// TwinCAT 3 PLC project TcoIo
// Title: TcoIo
// Company: Vortex.Library
// Author: Inxton
// ProjectVersion: 0.6.0.913
// ProgramVersion: 3.1.4023.0
// libraries:
//   Tc2_EtherCAT, * (Beckhoff Automation GmbH)
//   Tc2_Standard, * (Beckhoff Automation GmbH)
//   Tc2_System, * (Beckhoff Automation GmbH)
//   Tc3_Module, * (Beckhoff Automation GmbH)
//   TcoCore, 0.6.0.913 (Vortex.Library)
// project tree:
//   Diagnostics/EtherCAT/MasterDevice/Base/ EtcMasterBase_62654B43.TcDUT, SyncUnitsBase_AD6C35CE.TcDUT, SyncUnitTaskBase_FCD3CBF3.TcDUT, SyncUnitTasksBase_7C8711EB.TcDUT
//   Diagnostics/EtherCAT/MasterDevice/SyncUnit/ InfoData_8649EEEB.TcDUT, ITcoSyncUnit.TcIO, SyncUnitState.TcDUT, SyncUnitTask_AB2F5079.TcDUT, TcoSyncUnit.TcPOU
//   Diagnostics/EtherCAT/SlaveDevice/Base/ EtcSlaveBase_82538BE2.TcDUT, EtcSlaveBoxBase_77A0E4A7.TcDUT, EtcSlaveEndTerminalBase_866C7F0C.TcDUT, EtcSlaveTerminalBase_947E5A46.TcDUT
//   Diagnostics/EtherCAT/MasterDevice/ InfoData_84133AC9.TcDUT, Inputs_A65FACA4.TcDUT, Outputs_23C0ED1D.TcDUT, TcoEthercatDiagnosticsTask.TcPOU, TcoEthercatMasterDeviceState.TcDUT, ITcoEthercatMasterDevice.TcIO, TcoEthercatMasterDevice.TcPOU
//   Diagnostics/EtherCAT/MasterDevice/Messenger/ DiagnosticsMessenger.TcPOU, DiagnosticsMessengers.TcPOU
//   Diagnostics/EtherCAT/SlaveDevice/InfoData/ InfoData_23CBA837.TcDUT, InfoData_6F19DB2B.TcDUT
//   Diagnostics/EtherCAT/SlaveDevice/Inputs/ InputBase_8311D824.TcDUT
//   Diagnostics/EtherCAT/SlaveDevice/Outputs/ OutputBase_10CEE7DE.TcDUT
//   Diagnostics/EtherCAT/SlaveDevice/WcState/ WcState_0B2B16F9.TcDUT, WcState_9091E0EB.TcDUT
//   Diagnostics/EtherCAT/ TcoEthercat.TcGVL
//   Diagnostics/ProfinetComponent/ TcoPnIoComponent.TcPOU
//   EtherCAT/ eEcatState.TcDUT, eLinkState.TcDUT, ITcoEcatComponent.TcIO, TcoEcatSlaveState.TcPOU, TcoEcatComponent.TcPOU
//   / PlcTask.TcTTO
//   POUs/ MAIN.TcPOU
//   SpecialPlcTypes/ TcoAmsAddr.TcDUT, TcoAmsNetId.TcDUT
// real-time tasks:
//   TASK PlcTask: cycle T#10ms, priority 20, ADS port 350
//   TASK PlcTask1: cycle T#10ms, priority 21, ADS port 351
//   TASK PlcTask2: cycle T#10ms, priority 22, ADS port 352
// I/O:
//   DEVICE Device 1 (EtherCAT) (disabled), AmsNetId 172.20.10.104.2.1
//     Term 1 (EK1200) [EK1200-5000 EtherCAT Power supply (2A E-Bus)]
//       Term 2 (EL6002) [EL6002 Interface 2Ch. (RS232)]
//       Term 3 (EL1809) [EL1809 16Ch. Dig. Input 24V, 3ms]
//       Term 4 (EL2809) [EL2809 16Ch. Dig. Output 24V, 0.5A]
//       Term 5 (EL4004) [EL4004 4Ch. Ana. Output 0-10V, 12bit]
//       Term 6 (EL2809) [EL2809 16Ch. Dig. Output 24V, 0.5A]
//       Term 7 (EL6001) [EL6001 Interface (RS232)]
//       Term 8 (EL9011) [EL9011 End Terminal]
//   DEVICE Device 4 (EtherCAT) (disabled), AmsNetId 172.20.10.104.5.1
//     Term 9 (EK1100) [EK1100 EtherCAT Coupler (2A E-Bus)]
//       Term 10 (EK1122) [EK1122 2 port EtherCAT junction]
//         Term 11 (EK1100) [EK1100 EtherCAT Coupler (2A E-Bus)]
//           Term 12 (EL3174-0002) [EL3174-0002 4Ch. Ana. Input +/-10V, +/-20mA 16 Bit, Isolated Channels]
//           Term 13 (EL6001) [EL6001 Interface (RS232)]
//           Term 14 (EL3011) [EL3011 4Ch. Ana. Input 0-20mA DIFF]
//           Term 15 (EL2008) [EL2008 8Ch. Dig. Output 24V, 0.5A]
//           Term 16 (EL2008) [EL2008 8Ch. Dig. Output 24V, 0.5A]
//           Term 17 (EK1110) [EK1110 EtherCAT extension]
//         Term 18 (EK1100) [EK1100 EtherCAT Coupler (2A E-Bus)]
//           Term 19 (EL1809) [EL1809 16Ch. Dig. Input 24V, 3ms]
//           Term 20 (EL2809) [EL2809 16Ch. Dig. Output 24V, 0.5A]
//           Term 21 (EL1809) [EL1809 16Ch. Dig. Input 24V, 3ms]
//           Term 22 (EL3011) [EL3011 4Ch. Ana. Input 0-20mA DIFF]
//           Term 18 (EL9011) [EL9011 End Terminal]
//       Term 23 (EL3403) [EL3403 3Ch. Power Measuring]
//       Term 24 (EL6001) [EL6001 Interface (RS232)]
//       Term 25 (EL3024) [EL3024 4Ch. Ana. Input 4-20mA DIFF]
//       Term 19 (EL9011) [EL9011 End Terminal]
// variable links:
//   TcoIoTests/TcoIoTests Instance <-> Device 1 (EtherCAT)
//     PlcTask Inputs/GVL_iXlinker.Device_1_EtherCAT.InfoData.AmsNetId <-> InfoData/AmsNetId
//     PlcTask Inputs/GVL_iXlinker.Device_1_EtherCAT.InfoData.CfgSlaveCount <-> InfoData/CfgSlaveCount
//     PlcTask Inputs/GVL_iXlinker.Device_1_EtherCAT.InfoData.ChangeCount <-> InfoData/ChangeCount
//     PlcTask Inputs/GVL_iXlinker.Device_1_EtherCAT.InfoData.DevId <-> InfoData/DevId
//     PlcTask Inputs/GVL_iXlinker.Device_1_EtherCAT.Inputs.DevState <-> Inputs/DevState
//     PlcTask Inputs/GVL_iXlinker.Device_1_EtherCAT.Inputs.Frm0InputToggle <-> Inputs/Frm0InputToggle
//     PlcTask Inputs/GVL_iXlinker.Device_1_EtherCAT.Inputs.Frm0State <-> Inputs/Frm0State
//     PlcTask Inputs/GVL_iXlinker.Device_1_EtherCAT.Inputs.Frm0WcState <-> Inputs/Frm0WcState
//     PlcTask Inputs/GVL_iXlinker.Device_1_EtherCAT.Inputs.SlaveCount <-> Inputs/SlaveCount
//     PlcTask Inputs/GVL_iXlinker.Device_1_EtherCAT.SyncUnits._default.PlcTask1.InfoData.ObjectId <-> SyncUnits/<default>/PlcTask1/InfoData/ObjectId
//     PlcTask Inputs/GVL_iXlinker.Device_1_EtherCAT.SyncUnits._default.PlcTask1.InfoData.SlaveCount <-> SyncUnits/<default>/PlcTask1/InfoData/SlaveCount
//     PlcTask Inputs/GVL_iXlinker.Device_1_EtherCAT.SyncUnits._default.PlcTask1.InfoData.State <-> SyncUnits/<default>/PlcTask1/InfoData/State
//     PlcTask Inputs/GVL_iXlinker.Device_1_EtherCAT.SyncUnits._default.PlcTask1.WcState.WcState <-> SyncUnits/<default>/PlcTask1/WcState/WcState
//     PlcTask Outputs/GVL_iXlinker.Device_1_EtherCAT.Outputs.DevCtrl <-> Outputs/DevCtrl
//     PlcTask Outputs/GVL_iXlinker.Device_1_EtherCAT.Outputs.Frm0Ctrl <-> Outputs/Frm0Ctrl
//     PlcTask Outputs/GVL_iXlinker.Device_1_EtherCAT.Outputs.Frm0WcCtrl <-> Outputs/Frm0WcCtrl
//   TcoIoTests/TcoIoTests Instance <-> Device 1 (EtherCAT)/Term 1 (EK1200)/Term 2 (EL6002)
//     PlcTask Inputs/GVL_iXlinker.Device_1_EtherCAT.Term_1_EK1200.Term_2_EL6002.COM_TxPDO_Map_Inputs_Channel_1.Data_In[0] <-> COM TxPDO-Map Inputs Channel 1/Data In 0
//     PlcTask Inputs/GVL_iXlinker.Device_1_EtherCAT.Term_1_EK1200.Term_2_EL6002.COM_TxPDO_Map_Inputs_Channel_1.Data_In[10] <-> COM TxPDO-Map Inputs Channel 1/Data In 10
//     PlcTask Inputs/GVL_iXlinker.Device_1_EtherCAT.Term_1_EK1200.Term_2_EL6002.COM_TxPDO_Map_Inputs_Channel_1.Data_In[11] <-> COM TxPDO-Map Inputs Channel 1/Data In 11
//     PlcTask Inputs/GVL_iXlinker.Device_1_EtherCAT.Term_1_EK1200.Term_2_EL6002.COM_TxPDO_Map_Inputs_Channel_1.Data_In[12] <-> COM TxPDO-Map Inputs Channel 1/Data In 12
//     PlcTask Inputs/GVL_iXlinker.Device_1_EtherCAT.Term_1_EK1200.Term_2_EL6002.COM_TxPDO_Map_Inputs_Channel_1.Data_In[13] <-> COM TxPDO-Map Inputs Channel 1/Data In 13
//     PlcTask Inputs/GVL_iXlinker.Device_1_EtherCAT.Term_1_EK1200.Term_2_EL6002.COM_TxPDO_Map_Inputs_Channel_1.Data_In[14] <-> COM TxPDO-Map Inputs Channel 1/Data In 14
//     PlcTask Inputs/GVL_iXlinker.Device_1_EtherCAT.Term_1_EK1200.Term_2_EL6002.COM_TxPDO_Map_Inputs_Channel_1.Data_In[15] <-> COM TxPDO-Map Inputs Channel 1/Data In 15
//     PlcTask Inputs/GVL_iXlinker.Device_1_EtherCAT.Term_1_EK1200.Term_2_EL6002.COM_TxPDO_Map_Inputs_Channel_1.Data_In[16] <-> COM TxPDO-Map Inputs Channel 1/Data In 16
//     PlcTask Inputs/GVL_iXlinker.Device_1_EtherCAT.Term_1_EK1200.Term_2_EL6002.COM_TxPDO_Map_Inputs_Channel_1.Data_In[17] <-> COM TxPDO-Map Inputs Channel 1/Data In 17
//     PlcTask Inputs/GVL_iXlinker.Device_1_EtherCAT.Term_1_EK1200.Term_2_EL6002.COM_TxPDO_Map_Inputs_Channel_1.Data_In[18] <-> COM TxPDO-Map Inputs Channel 1/Data In 18
//     PlcTask Inputs/GVL_iXlinker.Device_1_EtherCAT.Term_1_EK1200.Term_2_EL6002.COM_TxPDO_Map_Inputs_Channel_1.Data_In[19] <-> COM TxPDO-Map Inputs Channel 1/Data In 19
//     PlcTask Inputs/GVL_iXlinker.Device_1_EtherCAT.Term_1_EK1200.Term_2_EL6002.COM_TxPDO_Map_Inputs_Channel_1.Data_In[1] <-> COM TxPDO-Map Inputs Channel 1/Data In 1
//     PlcTask Inputs/GVL_iXlinker.Device_1_EtherCAT.Term_1_EK1200.Term_2_EL6002.COM_TxPDO_Map_Inputs_Channel_1.Data_In[20] <-> COM TxPDO-Map Inputs Channel 1/Data In 20
//     PlcTask Inputs/GVL_iXlinker.Device_1_EtherCAT.Term_1_EK1200.Term_2_EL6002.COM_TxPDO_Map_Inputs_Channel_1.Data_In[21] <-> COM TxPDO-Map Inputs Channel 1/Data In 21
//     PlcTask Inputs/GVL_iXlinker.Device_1_EtherCAT.Term_1_EK1200.Term_2_EL6002.COM_TxPDO_Map_Inputs_Channel_1.Data_In[2] <-> COM TxPDO-Map Inputs Channel 1/Data In 2
//     PlcTask Inputs/GVL_iXlinker.Device_1_EtherCAT.Term_1_EK1200.Term_2_EL6002.COM_TxPDO_Map_Inputs_Channel_1.Data_In[3] <-> COM TxPDO-Map Inputs Channel 1/Data In 3
//     PlcTask Inputs/GVL_iXlinker.Device_1_EtherCAT.Term_1_EK1200.Term_2_EL6002.COM_TxPDO_Map_Inputs_Channel_1.Data_In[4] <-> COM TxPDO-Map Inputs Channel 1/Data In 4
//     PlcTask Inputs/GVL_iXlinker.Device_1_EtherCAT.Term_1_EK1200.Term_2_EL6002.COM_TxPDO_Map_Inputs_Channel_1.Data_In[5] <-> COM TxPDO-Map Inputs Channel 1/Data In 5
//     PlcTask Inputs/GVL_iXlinker.Device_1_EtherCAT.Term_1_EK1200.Term_2_EL6002.COM_TxPDO_Map_Inputs_Channel_1.Data_In[6] <-> COM TxPDO-Map Inputs Channel 1/Data In 6
//     PlcTask Inputs/GVL_iXlinker.Device_1_EtherCAT.Term_1_EK1200.Term_2_EL6002.COM_TxPDO_Map_Inputs_Channel_1.Data_In[7] <-> COM TxPDO-Map Inputs Channel 1/Data In 7
//     PlcTask Inputs/GVL_iXlinker.Device_1_EtherCAT.Term_1_EK1200.Term_2_EL6002.COM_TxPDO_Map_Inputs_Channel_1.Data_In[8] <-> COM TxPDO-Map Inputs Channel 1/Data In 8
//     PlcTask Inputs/GVL_iXlinker.Device_1_EtherCAT.Term_1_EK1200.Term_2_EL6002.COM_TxPDO_Map_Inputs_Channel_1.Data_In[9] <-> COM TxPDO-Map Inputs Channel 1/Data In 9
//     PlcTask Inputs/GVL_iXlinker.Device_1_EtherCAT.Term_1_EK1200.Term_2_EL6002.COM_TxPDO_Map_Inputs_Channel_2.Data_In[0] <-> COM TxPDO-Map Inputs Channel 2/Data In 0
//     PlcTask Inputs/GVL_iXlinker.Device_1_EtherCAT.Term_1_EK1200.Term_2_EL6002.COM_TxPDO_Map_Inputs_Channel_2.Data_In[10] <-> COM TxPDO-Map Inputs Channel 2/Data In 10
//     PlcTask Inputs/GVL_iXlinker.Device_1_EtherCAT.Term_1_EK1200.Term_2_EL6002.COM_TxPDO_Map_Inputs_Channel_2.Data_In[11] <-> COM TxPDO-Map Inputs Channel 2/Data In 11
//     PlcTask Inputs/GVL_iXlinker.Device_1_EtherCAT.Term_1_EK1200.Term_2_EL6002.COM_TxPDO_Map_Inputs_Channel_2.Data_In[12] <-> COM TxPDO-Map Inputs Channel 2/Data In 12
//     PlcTask Inputs/GVL_iXlinker.Device_1_EtherCAT.Term_1_EK1200.Term_2_EL6002.COM_TxPDO_Map_Inputs_Channel_2.Data_In[13] <-> COM TxPDO-Map Inputs Channel 2/Data In 13
//     PlcTask Inputs/GVL_iXlinker.Device_1_EtherCAT.Term_1_EK1200.Term_2_EL6002.COM_TxPDO_Map_Inputs_Channel_2.Data_In[14] <-> COM TxPDO-Map Inputs Channel 2/Data In 14
//     PlcTask Inputs/GVL_iXlinker.Device_1_EtherCAT.Term_1_EK1200.Term_2_EL6002.COM_TxPDO_Map_Inputs_Channel_2.Data_In[15] <-> COM TxPDO-Map Inputs Channel 2/Data In 15
//     PlcTask Inputs/GVL_iXlinker.Device_1_EtherCAT.Term_1_EK1200.Term_2_EL6002.COM_TxPDO_Map_Inputs_Channel_2.Data_In[16] <-> COM TxPDO-Map Inputs Channel 2/Data In 16
//     PlcTask Inputs/GVL_iXlinker.Device_1_EtherCAT.Term_1_EK1200.Term_2_EL6002.COM_TxPDO_Map_Inputs_Channel_2.Data_In[17] <-> COM TxPDO-Map Inputs Channel 2/Data In 17
//     PlcTask Inputs/GVL_iXlinker.Device_1_EtherCAT.Term_1_EK1200.Term_2_EL6002.COM_TxPDO_Map_Inputs_Channel_2.Data_In[18] <-> COM TxPDO-Map Inputs Channel 2/Data In 18
//     PlcTask Inputs/GVL_iXlinker.Device_1_EtherCAT.Term_1_EK1200.Term_2_EL6002.COM_TxPDO_Map_Inputs_Channel_2.Data_In[19] <-> COM TxPDO-Map Inputs Channel 2/Data In 19
//     PlcTask Inputs/GVL_iXlinker.Device_1_EtherCAT.Term_1_EK1200.Term_2_EL6002.COM_TxPDO_Map_Inputs_Channel_2.Data_In[1] <-> COM TxPDO-Map Inputs Channel 2/Data In 1
//     PlcTask Inputs/GVL_iXlinker.Device_1_EtherCAT.Term_1_EK1200.Term_2_EL6002.COM_TxPDO_Map_Inputs_Channel_2.Data_In[20] <-> COM TxPDO-Map Inputs Channel 2/Data In 20
//     PlcTask Inputs/GVL_iXlinker.Device_1_EtherCAT.Term_1_EK1200.Term_2_EL6002.COM_TxPDO_Map_Inputs_Channel_2.Data_In[21] <-> COM TxPDO-Map Inputs Channel 2/Data In 21
//     PlcTask Inputs/GVL_iXlinker.Device_1_EtherCAT.Term_1_EK1200.Term_2_EL6002.COM_TxPDO_Map_Inputs_Channel_2.Data_In[2] <-> COM TxPDO-Map Inputs Channel 2/Data In 2
//     PlcTask Inputs/GVL_iXlinker.Device_1_EtherCAT.Term_1_EK1200.Term_2_EL6002.COM_TxPDO_Map_Inputs_Channel_2.Data_In[3] <-> COM TxPDO-Map Inputs Channel 2/Data In 3
//     PlcTask Inputs/GVL_iXlinker.Device_1_EtherCAT.Term_1_EK1200.Term_2_EL6002.COM_TxPDO_Map_Inputs_Channel_2.Data_In[4] <-> COM TxPDO-Map Inputs Channel 2/Data In 4
//     PlcTask Inputs/GVL_iXlinker.Device_1_EtherCAT.Term_1_EK1200.Term_2_EL6002.COM_TxPDO_Map_Inputs_Channel_2.Data_In[5] <-> COM TxPDO-Map Inputs Channel 2/Data In 5
//     PlcTask Inputs/GVL_iXlinker.Device_1_EtherCAT.Term_1_EK1200.Term_2_EL6002.COM_TxPDO_Map_Inputs_Channel_2.Data_In[6] <-> COM TxPDO-Map Inputs Channel 2/Data In 6
//     PlcTask Inputs/GVL_iXlinker.Device_1_EtherCAT.Term_1_EK1200.Term_2_EL6002.COM_TxPDO_Map_Inputs_Channel_2.Data_In[7] <-> COM TxPDO-Map Inputs Channel 2/Data In 7
//     PlcTask Inputs/GVL_iXlinker.Device_1_EtherCAT.Term_1_EK1200.Term_2_EL6002.COM_TxPDO_Map_Inputs_Channel_2.Data_In[8] <-> COM TxPDO-Map Inputs Channel 2/Data In 8
//     PlcTask Inputs/GVL_iXlinker.Device_1_EtherCAT.Term_1_EK1200.Term_2_EL6002.COM_TxPDO_Map_Inputs_Channel_2.Data_In[9] <-> COM TxPDO-Map Inputs Channel 2/Data In 9
//     PlcTask Inputs/GVL_iXlinker.Device_1_EtherCAT.Term_1_EK1200.Term_2_EL6002.COM_TxPDO_Map_Inputs_Channel_1.Status/Buffer_full <-> COM TxPDO-Map Inputs Channel 1/Status/Buffer full
//     PlcTask Inputs/GVL_iXlinker.Device_1_EtherCAT.Term_1_EK1200.Term_2_EL6002.COM_TxPDO_Map_Inputs_Channel_2.Status/Buffer_full <-> COM TxPDO-Map Inputs Channel 2/Status/Buffer full
//     PlcTask Inputs/GVL_iXlinker.Device_1_EtherCAT.Term_1_EK1200.Term_2_EL6002.COM_TxPDO_Map_Inputs_Channel_1.Status/Framing_error <-> COM TxPDO-Map Inputs Channel 1/Status/Framing error
//     PlcTask Inputs/GVL_iXlinker.Device_1_EtherCAT.Term_1_EK1200.Term_2_EL6002.COM_TxPDO_Map_Inputs_Channel_2.Status/Framing_error <-> COM TxPDO-Map Inputs Channel 2/Status/Framing error
//     PlcTask Inputs/GVL_iXlinker.Device_1_EtherCAT.Term_1_EK1200.Term_2_EL6002.COM_TxPDO_Map_Inputs_Channel_1.Status/Init_accepted <-> COM TxPDO-Map Inputs Channel 1/Status/Init accepted
//     PlcTask Inputs/GVL_iXlinker.Device_1_EtherCAT.Term_1_EK1200.Term_2_EL6002.COM_TxPDO_Map_Inputs_Channel_2.Status/Init_accepted <-> COM TxPDO-Map Inputs Channel 2/Status/Init accepted
//     PlcTask Inputs/GVL_iXlinker.Device_1_EtherCAT.Term_1_EK1200.Term_2_EL6002.COM_TxPDO_Map_Inputs_Channel_1.Status/Input_length <-> COM TxPDO-Map Inputs Channel 1/Status/Input length
//     PlcTask Inputs/GVL_iXlinker.Device_1_EtherCAT.Term_1_EK1200.Term_2_EL6002.COM_TxPDO_Map_Inputs_Channel_2.Status/Input_length <-> COM TxPDO-Map Inputs Channel 2/Status/Input length
//     PlcTask Inputs/GVL_iXlinker.Device_1_EtherCAT.Term_1_EK1200.Term_2_EL6002.COM_TxPDO_Map_Inputs_Channel_1.Status/Overrun_error <-> COM TxPDO-Map Inputs Channel 1/Status/Overrun error
//     PlcTask Inputs/GVL_iXlinker.Device_1_EtherCAT.Term_1_EK1200.Term_2_EL6002.COM_TxPDO_Map_Inputs_Channel_2.Status/Overrun_error <-> COM TxPDO-Map Inputs Channel 2/Status/Overrun error
//     PlcTask Inputs/GVL_iXlinker.Device_1_EtherCAT.Term_1_EK1200.Term_2_EL6002.COM_TxPDO_Map_Inputs_Channel_1.Status/Parity_error <-> COM TxPDO-Map Inputs Channel 1/Status/Parity error
//     PlcTask Inputs/GVL_iXlinker.Device_1_EtherCAT.Term_1_EK1200.Term_2_EL6002.COM_TxPDO_Map_Inputs_Channel_2.Status/Parity_error <-> COM TxPDO-Map Inputs Channel 2/Status/Parity error
//     PlcTask Inputs/GVL_iXlinker.Device_1_EtherCAT.Term_1_EK1200.Term_2_EL6002.COM_TxPDO_Map_Inputs_Channel_1.Status/Receive_request <-> COM TxPDO-Map Inputs Channel 1/Status/Receive request
//     PlcTask Inputs/GVL_iXlinker.Device_1_EtherCAT.Term_1_EK1200.Term_2_EL6002.COM_TxPDO_Map_Inputs_Channel_2.Status/Receive_request <-> COM TxPDO-Map Inputs Channel 2/Status/Receive request
//     PlcTask Inputs/GVL_iXlinker.Device_1_EtherCAT.Term_1_EK1200.Term_2_EL6002.COM_TxPDO_Map_Inputs_Channel_1.Status/Transmit_accepted <-> COM TxPDO-Map Inputs Channel 1/Status/Transmit accepted
//     PlcTask Inputs/GVL_iXlinker.Device_1_EtherCAT.Term_1_EK1200.Term_2_EL6002.COM_TxPDO_Map_Inputs_Channel_2.Status/Transmit_accepted <-> COM TxPDO-Map Inputs Channel 2/Status/Transmit accepted
//     PlcTask Inputs/GVL_iXlinker.Device_1_EtherCAT.Term_1_EK1200.Term_2_EL6002.InfoData.AdsAddr <-> InfoData/AdsAddr
//     PlcTask Inputs/GVL_iXlinker.Device_1_EtherCAT.Term_1_EK1200.Term_2_EL6002.InfoData.State <-> InfoData/State
//     PlcTask Inputs/GVL_iXlinker.Device_1_EtherCAT.Term_1_EK1200.Term_2_EL6002.WcState.InputToggle <-> WcState/InputToggle
//     PlcTask Inputs/GVL_iXlinker.Device_1_EtherCAT.Term_1_EK1200.Term_2_EL6002.WcState.WcState <-> WcState/WcState
//     PlcTask Outputs/GVL_iXlinker.Device_1_EtherCAT.Term_1_EK1200.Term_2_EL6002.COM_RxPDO_Map_Outputs_Channel_1.Ctrl/Init_request <-> COM RxPDO-Map Outputs Channel 1/Ctrl/Init request
//     PlcTask Outputs/GVL_iXlinker.Device_1_EtherCAT.Term_1_EK1200.Term_2_EL6002.COM_RxPDO_Map_Outputs_Channel_2.Ctrl/Init_request <-> COM RxPDO-Map Outputs Channel 2/Ctrl/Init request
//     PlcTask Outputs/GVL_iXlinker.Device_1_EtherCAT.Term_1_EK1200.Term_2_EL6002.COM_RxPDO_Map_Outputs_Channel_1.Ctrl/Output_length <-> COM RxPDO-Map Outputs Channel 1/Ctrl/Output length
//     PlcTask Outputs/GVL_iXlinker.Device_1_EtherCAT.Term_1_EK1200.Term_2_EL6002.COM_RxPDO_Map_Outputs_Channel_2.Ctrl/Output_length <-> COM RxPDO-Map Outputs Channel 2/Ctrl/Output length
//     PlcTask Outputs/GVL_iXlinker.Device_1_EtherCAT.Term_1_EK1200.Term_2_EL6002.COM_RxPDO_Map_Outputs_Channel_1.Ctrl/Receive_accepted <-> COM RxPDO-Map Outputs Channel 1/Ctrl/Receive accepted
//     PlcTask Outputs/GVL_iXlinker.Device_1_EtherCAT.Term_1_EK1200.Term_2_EL6002.COM_RxPDO_Map_Outputs_Channel_2.Ctrl/Receive_accepted <-> COM RxPDO-Map Outputs Channel 2/Ctrl/Receive accepted
//     PlcTask Outputs/GVL_iXlinker.Device_1_EtherCAT.Term_1_EK1200.Term_2_EL6002.COM_RxPDO_Map_Outputs_Channel_1.Ctrl/Send_continuous <-> COM RxPDO-Map Outputs Channel 1/Ctrl/Send continuous
//     PlcTask Outputs/GVL_iXlinker.Device_1_EtherCAT.Term_1_EK1200.Term_2_EL6002.COM_RxPDO_Map_Outputs_Channel_2.Ctrl/Send_continuous <-> COM RxPDO-Map Outputs Channel 2/Ctrl/Send continuous
//     PlcTask Outputs/GVL_iXlinker.Device_1_EtherCAT.Term_1_EK1200.Term_2_EL6002.COM_RxPDO_Map_Outputs_Channel_1.Ctrl/Transmit_request <-> COM RxPDO-Map Outputs Channel 1/Ctrl/Transmit request
//     PlcTask Outputs/GVL_iXlinker.Device_1_EtherCAT.Term_1_EK1200.Term_2_EL6002.COM_RxPDO_Map_Outputs_Channel_2.Ctrl/Transmit_request <-> COM RxPDO-Map Outputs Channel 2/Ctrl/Transmit request
//     PlcTask Outputs/GVL_iXlinker.Device_1_EtherCAT.Term_1_EK1200.Term_2_EL6002.COM_RxPDO_Map_Outputs_Channel_1.Data_Out[0] <-> COM RxPDO-Map Outputs Channel 1/Data Out 0
//     PlcTask Outputs/GVL_iXlinker.Device_1_EtherCAT.Term_1_EK1200.Term_2_EL6002.COM_RxPDO_Map_Outputs_Channel_1.Data_Out[10] <-> COM RxPDO-Map Outputs Channel 1/Data Out 10
//     PlcTask Outputs/GVL_iXlinker.Device_1_EtherCAT.Term_1_EK1200.Term_2_EL6002.COM_RxPDO_Map_Outputs_Channel_1.Data_Out[11] <-> COM RxPDO-Map Outputs Channel 1/Data Out 11
//     PlcTask Outputs/GVL_iXlinker.Device_1_EtherCAT.Term_1_EK1200.Term_2_EL6002.COM_RxPDO_Map_Outputs_Channel_1.Data_Out[12] <-> COM RxPDO-Map Outputs Channel 1/Data Out 12
//     PlcTask Outputs/GVL_iXlinker.Device_1_EtherCAT.Term_1_EK1200.Term_2_EL6002.COM_RxPDO_Map_Outputs_Channel_1.Data_Out[13] <-> COM RxPDO-Map Outputs Channel 1/Data Out 13
//     PlcTask Outputs/GVL_iXlinker.Device_1_EtherCAT.Term_1_EK1200.Term_2_EL6002.COM_RxPDO_Map_Outputs_Channel_1.Data_Out[14] <-> COM RxPDO-Map Outputs Channel 1/Data Out 14
//     PlcTask Outputs/GVL_iXlinker.Device_1_EtherCAT.Term_1_EK1200.Term_2_EL6002.COM_RxPDO_Map_Outputs_Channel_1.Data_Out[15] <-> COM RxPDO-Map Outputs Channel 1/Data Out 15
//     PlcTask Outputs/GVL_iXlinker.Device_1_EtherCAT.Term_1_EK1200.Term_2_EL6002.COM_RxPDO_Map_Outputs_Channel_1.Data_Out[16] <-> COM RxPDO-Map Outputs Channel 1/Data Out 16
//     PlcTask Outputs/GVL_iXlinker.Device_1_EtherCAT.Term_1_EK1200.Term_2_EL6002.COM_RxPDO_Map_Outputs_Channel_1.Data_Out[17] <-> COM RxPDO-Map Outputs Channel 1/Data Out 17
//     PlcTask Outputs/GVL_iXlinker.Device_1_EtherCAT.Term_1_EK1200.Term_2_EL6002.COM_RxPDO_Map_Outputs_Channel_1.Data_Out[18] <-> COM RxPDO-Map Outputs Channel 1/Data Out 18
//     PlcTask Outputs/GVL_iXlinker.Device_1_EtherCAT.Term_1_EK1200.Term_2_EL6002.COM_RxPDO_Map_Outputs_Channel_1.Data_Out[19] <-> COM RxPDO-Map Outputs Channel 1/Data Out 19
//     PlcTask Outputs/GVL_iXlinker.Device_1_EtherCAT.Term_1_EK1200.Term_2_EL6002.COM_RxPDO_Map_Outputs_Channel_1.Data_Out[1] <-> COM RxPDO-Map Outputs Channel 1/Data Out 1
//     PlcTask Outputs/GVL_iXlinker.Device_1_EtherCAT.Term_1_EK1200.Term_2_EL6002.COM_RxPDO_Map_Outputs_Channel_1.Data_Out[20] <-> COM RxPDO-Map Outputs Channel 1/Data Out 20
//     PlcTask Outputs/GVL_iXlinker.Device_1_EtherCAT.Term_1_EK1200.Term_2_EL6002.COM_RxPDO_Map_Outputs_Channel_1.Data_Out[21] <-> COM RxPDO-Map Outputs Channel 1/Data Out 21
//     PlcTask Outputs/GVL_iXlinker.Device_1_EtherCAT.Term_1_EK1200.Term_2_EL6002.COM_RxPDO_Map_Outputs_Channel_1.Data_Out[2] <-> COM RxPDO-Map Outputs Channel 1/Data Out 2
//     PlcTask Outputs/GVL_iXlinker.Device_1_EtherCAT.Term_1_EK1200.Term_2_EL6002.COM_RxPDO_Map_Outputs_Channel_1.Data_Out[3] <-> COM RxPDO-Map Outputs Channel 1/Data Out 3
//     PlcTask Outputs/GVL_iXlinker.Device_1_EtherCAT.Term_1_EK1200.Term_2_EL6002.COM_RxPDO_Map_Outputs_Channel_1.Data_Out[4] <-> COM RxPDO-Map Outputs Channel 1/Data Out 4
//     PlcTask Outputs/GVL_iXlinker.Device_1_EtherCAT.Term_1_EK1200.Term_2_EL6002.COM_RxPDO_Map_Outputs_Channel_1.Data_Out[5] <-> COM RxPDO-Map Outputs Channel 1/Data Out 5
//     PlcTask Outputs/GVL_iXlinker.Device_1_EtherCAT.Term_1_EK1200.Term_2_EL6002.COM_RxPDO_Map_Outputs_Channel_1.Data_Out[6] <-> COM RxPDO-Map Outputs Channel 1/Data Out 6
//     PlcTask Outputs/GVL_iXlinker.Device_1_EtherCAT.Term_1_EK1200.Term_2_EL6002.COM_RxPDO_Map_Outputs_Channel_1.Data_Out[7] <-> COM RxPDO-Map Outputs Channel 1/Data Out 7
//     PlcTask Outputs/GVL_iXlinker.Device_1_EtherCAT.Term_1_EK1200.Term_2_EL6002.COM_RxPDO_Map_Outputs_Channel_1.Data_Out[8] <-> COM RxPDO-Map Outputs Channel 1/Data Out 8
//     PlcTask Outputs/GVL_iXlinker.Device_1_EtherCAT.Term_1_EK1200.Term_2_EL6002.COM_RxPDO_Map_Outputs_Channel_1.Data_Out[9] <-> COM RxPDO-Map Outputs Channel 1/Data Out 9
//     PlcTask Outputs/GVL_iXlinker.Device_1_EtherCAT.Term_1_EK1200.Term_2_EL6002.COM_RxPDO_Map_Outputs_Channel_2.Data_Out[0] <-> COM RxPDO-Map Outputs Channel 2/Data Out 0
//     PlcTask Outputs/GVL_iXlinker.Device_1_EtherCAT.Term_1_EK1200.Term_2_EL6002.COM_RxPDO_Map_Outputs_Channel_2.Data_Out[10] <-> COM RxPDO-Map Outputs Channel 2/Data Out 10
//     PlcTask Outputs/GVL_iXlinker.Device_1_EtherCAT.Term_1_EK1200.Term_2_EL6002.COM_RxPDO_Map_Outputs_Channel_2.Data_Out[11] <-> COM RxPDO-Map Outputs Channel 2/Data Out 11
//     PlcTask Outputs/GVL_iXlinker.Device_1_EtherCAT.Term_1_EK1200.Term_2_EL6002.COM_RxPDO_Map_Outputs_Channel_2.Data_Out[12] <-> COM RxPDO-Map Outputs Channel 2/Data Out 12
//     PlcTask Outputs/GVL_iXlinker.Device_1_EtherCAT.Term_1_EK1200.Term_2_EL6002.COM_RxPDO_Map_Outputs_Channel_2.Data_Out[13] <-> COM RxPDO-Map Outputs Channel 2/Data Out 13
//     PlcTask Outputs/GVL_iXlinker.Device_1_EtherCAT.Term_1_EK1200.Term_2_EL6002.COM_RxPDO_Map_Outputs_Channel_2.Data_Out[14] <-> COM RxPDO-Map Outputs Channel 2/Data Out 14
//     PlcTask Outputs/GVL_iXlinker.Device_1_EtherCAT.Term_1_EK1200.Term_2_EL6002.COM_RxPDO_Map_Outputs_Channel_2.Data_Out[15] <-> COM RxPDO-Map Outputs Channel 2/Data Out 15
//     PlcTask Outputs/GVL_iXlinker.Device_1_EtherCAT.Term_1_EK1200.Term_2_EL6002.COM_RxPDO_Map_Outputs_Channel_2.Data_Out[16] <-> COM RxPDO-Map Outputs Channel 2/Data Out 16
//     PlcTask Outputs/GVL_iXlinker.Device_1_EtherCAT.Term_1_EK1200.Term_2_EL6002.COM_RxPDO_Map_Outputs_Channel_2.Data_Out[17] <-> COM RxPDO-Map Outputs Channel 2/Data Out 17
//     PlcTask Outputs/GVL_iXlinker.Device_1_EtherCAT.Term_1_EK1200.Term_2_EL6002.COM_RxPDO_Map_Outputs_Channel_2.Data_Out[18] <-> COM RxPDO-Map Outputs Channel 2/Data Out 18
//     PlcTask Outputs/GVL_iXlinker.Device_1_EtherCAT.Term_1_EK1200.Term_2_EL6002.COM_RxPDO_Map_Outputs_Channel_2.Data_Out[19] <-> COM RxPDO-Map Outputs Channel 2/Data Out 19
//     PlcTask Outputs/GVL_iXlinker.Device_1_EtherCAT.Term_1_EK1200.Term_2_EL6002.COM_RxPDO_Map_Outputs_Channel_2.Data_Out[1] <-> COM RxPDO-Map Outputs Channel 2/Data Out 1
//     PlcTask Outputs/GVL_iXlinker.Device_1_EtherCAT.Term_1_EK1200.Term_2_EL6002.COM_RxPDO_Map_Outputs_Channel_2.Data_Out[20] <-> COM RxPDO-Map Outputs Channel 2/Data Out 20
//     PlcTask Outputs/GVL_iXlinker.Device_1_EtherCAT.Term_1_EK1200.Term_2_EL6002.COM_RxPDO_Map_Outputs_Channel_2.Data_Out[21] <-> COM RxPDO-Map Outputs Channel 2/Data Out 21
//     PlcTask Outputs/GVL_iXlinker.Device_1_EtherCAT.Term_1_EK1200.Term_2_EL6002.COM_RxPDO_Map_Outputs_Channel_2.Data_Out[2] <-> COM RxPDO-Map Outputs Channel 2/Data Out 2
//     PlcTask Outputs/GVL_iXlinker.Device_1_EtherCAT.Term_1_EK1200.Term_2_EL6002.COM_RxPDO_Map_Outputs_Channel_2.Data_Out[3] <-> COM RxPDO-Map Outputs Channel 2/Data Out 3
//     PlcTask Outputs/GVL_iXlinker.Device_1_EtherCAT.Term_1_EK1200.Term_2_EL6002.COM_RxPDO_Map_Outputs_Channel_2.Data_Out[4] <-> COM RxPDO-Map Outputs Channel 2/Data Out 4
//     PlcTask Outputs/GVL_iXlinker.Device_1_EtherCAT.Term_1_EK1200.Term_2_EL6002.COM_RxPDO_Map_Outputs_Channel_2.Data_Out[5] <-> COM RxPDO-Map Outputs Channel 2/Data Out 5
//     PlcTask Outputs/GVL_iXlinker.Device_1_EtherCAT.Term_1_EK1200.Term_2_EL6002.COM_RxPDO_Map_Outputs_Channel_2.Data_Out[6] <-> COM RxPDO-Map Outputs Channel 2/Data Out 6
//     PlcTask Outputs/GVL_iXlinker.Device_1_EtherCAT.Term_1_EK1200.Term_2_EL6002.COM_RxPDO_Map_Outputs_Channel_2.Data_Out[7] <-> COM RxPDO-Map Outputs Channel 2/Data Out 7
//     PlcTask Outputs/GVL_iXlinker.Device_1_EtherCAT.Term_1_EK1200.Term_2_EL6002.COM_RxPDO_Map_Outputs_Channel_2.Data_Out[8] <-> COM RxPDO-Map Outputs Channel 2/Data Out 8
//     PlcTask Outputs/GVL_iXlinker.Device_1_EtherCAT.Term_1_EK1200.Term_2_EL6002.COM_RxPDO_Map_Outputs_Channel_2.Data_Out[9] <-> COM RxPDO-Map Outputs Channel 2/Data Out 9
//   TcoIoTests/TcoIoTests Instance <-> Device 1 (EtherCAT)/Term 1 (EK1200)/Term 3 (EL1809)
//     PlcTask Inputs/GVL_iXlinker.Device_1_EtherCAT.Term_1_EK1200.Term_3_EL1809.Channel_{1..16}.Input <-> Channel {1..16}/Input  (16 links)
//     PlcTask Inputs/GVL_iXlinker.Device_1_EtherCAT.Term_1_EK1200.Term_3_EL1809.InfoData.State <-> InfoData/State
//     PlcTask Inputs/GVL_iXlinker.Device_1_EtherCAT.Term_1_EK1200.Term_3_EL1809.WcState.InputToggle <-> WcState/InputToggle
//     PlcTask Inputs/GVL_iXlinker.Device_1_EtherCAT.Term_1_EK1200.Term_3_EL1809.WcState.WcState <-> WcState/WcState
//   TcoIoTests/TcoIoTests Instance <-> Device 1 (EtherCAT)/Term 1 (EK1200)/Term 4 (EL2809)
//     PlcTask Inputs/GVL_iXlinker.Device_1_EtherCAT.Term_1_EK1200.Term_4_EL2809.InfoData.State <-> InfoData/State
//     PlcTask Inputs/GVL_iXlinker.Device_1_EtherCAT.Term_1_EK1200.Term_4_EL2809.WcState.WcState <-> WcState/WcState
//     PlcTask Outputs/GVL_iXlinker.Device_1_EtherCAT.Term_1_EK1200.Term_4_EL2809.Channel_{1..16}.Output <-> Channel {1..16}/Output  (16 links)
//   TcoIoTests/TcoIoTests Instance <-> Device 1 (EtherCAT)/Term 1 (EK1200)/Term 5 (EL4004)
//     PlcTask Inputs/GVL_iXlinker.Device_1_EtherCAT.Term_1_EK1200.Term_5_EL4004.InfoData.AdsAddr <-> InfoData/AdsAddr
//     PlcTask Inputs/GVL_iXlinker.Device_1_EtherCAT.Term_1_EK1200.Term_5_EL4004.InfoData.State <-> InfoData/State
//     PlcTask Inputs/GVL_iXlinker.Device_1_EtherCAT.Term_1_EK1200.Term_5_EL4004.WcState.WcState <-> WcState/WcState
//     PlcTask Outputs/GVL_iXlinker.Device_1_EtherCAT.Term_1_EK1200.Term_5_EL4004.AO_Outputs_Channel_{1..4}.Analog_output <-> AO Outputs Channel {1..4}/Analog output  (4 links)
//   TcoIoTests/TcoIoTests Instance <-> Device 1 (EtherCAT)/Term 1 (EK1200)/Term 6 (EL2809)
//     PlcTask Inputs/GVL_iXlinker.Device_1_EtherCAT.Term_1_EK1200.Term_6_EL2809.InfoData.State <-> InfoData/State
//     PlcTask Inputs/GVL_iXlinker.Device_1_EtherCAT.Term_1_EK1200.Term_6_EL2809.WcState.WcState <-> WcState/WcState
//     PlcTask Outputs/GVL_iXlinker.Device_1_EtherCAT.Term_1_EK1200.Term_6_EL2809.Channel_{1..16}.Output <-> Channel {1..16}/Output  (16 links)
//   TcoIoTests/TcoIoTests Instance <-> Device 1 (EtherCAT)/Term 1 (EK1200)/Term 7 (EL6001)
//     PlcTask Inputs/GVL_iXlinker.Device_1_EtherCAT.Term_1_EK1200.Term_7_EL6001.COM_Inputs.Data_In[{0..21}] <-> COM Inputs/Data In {0..21}  (22 links)
//     PlcTask Inputs/GVL_iXlinker.Device_1_EtherCAT.Term_1_EK1200.Term_7_EL6001.COM_Inputs.Status/Buffer_full <-> COM Inputs/Status/Buffer full
//     PlcTask Inputs/GVL_iXlinker.Device_1_EtherCAT.Term_1_EK1200.Term_7_EL6001.COM_Inputs.Status/Framing_error <-> COM Inputs/Status/Framing error
//     PlcTask Inputs/GVL_iXlinker.Device_1_EtherCAT.Term_1_EK1200.Term_7_EL6001.COM_Inputs.Status/Init_accepted <-> COM Inputs/Status/Init accepted
//     PlcTask Inputs/GVL_iXlinker.Device_1_EtherCAT.Term_1_EK1200.Term_7_EL6001.COM_Inputs.Status/Input_length <-> COM Inputs/Status/Input length
//     PlcTask Inputs/GVL_iXlinker.Device_1_EtherCAT.Term_1_EK1200.Term_7_EL6001.COM_Inputs.Status/Overrun_error <-> COM Inputs/Status/Overrun error
//     PlcTask Inputs/GVL_iXlinker.Device_1_EtherCAT.Term_1_EK1200.Term_7_EL6001.COM_Inputs.Status/Parity_error <-> COM Inputs/Status/Parity error
//     PlcTask Inputs/GVL_iXlinker.Device_1_EtherCAT.Term_1_EK1200.Term_7_EL6001.COM_Inputs.Status/Receive_request <-> COM Inputs/Status/Receive request
//     PlcTask Inputs/GVL_iXlinker.Device_1_EtherCAT.Term_1_EK1200.Term_7_EL6001.COM_Inputs.Status/Transmit_accepted <-> COM Inputs/Status/Transmit accepted
//     PlcTask Inputs/GVL_iXlinker.Device_1_EtherCAT.Term_1_EK1200.Term_7_EL6001.InfoData.AdsAddr <-> InfoData/AdsAddr
//     PlcTask Inputs/GVL_iXlinker.Device_1_EtherCAT.Term_1_EK1200.Term_7_EL6001.InfoData.State <-> InfoData/State
//     PlcTask Inputs/GVL_iXlinker.Device_1_EtherCAT.Term_1_EK1200.Term_7_EL6001.WcState.InputToggle <-> WcState/InputToggle
//     PlcTask Inputs/GVL_iXlinker.Device_1_EtherCAT.Term_1_EK1200.Term_7_EL6001.WcState.WcState <-> WcState/WcState
//     PlcTask Outputs/GVL_iXlinker.Device_1_EtherCAT.Term_1_EK1200.Term_7_EL6001.COM_Outputs.Ctrl/Init_request <-> COM Outputs/Ctrl/Init request
//     PlcTask Outputs/GVL_iXlinker.Device_1_EtherCAT.Term_1_EK1200.Term_7_EL6001.COM_Outputs.Ctrl/Output_length <-> COM Outputs/Ctrl/Output length
//     PlcTask Outputs/GVL_iXlinker.Device_1_EtherCAT.Term_1_EK1200.Term_7_EL6001.COM_Outputs.Ctrl/Receive_accepted <-> COM Outputs/Ctrl/Receive accepted
//     PlcTask Outputs/GVL_iXlinker.Device_1_EtherCAT.Term_1_EK1200.Term_7_EL6001.COM_Outputs.Ctrl/Send_continues <-> COM Outputs/Ctrl/Send continues
//     PlcTask Outputs/GVL_iXlinker.Device_1_EtherCAT.Term_1_EK1200.Term_7_EL6001.COM_Outputs.Ctrl/Transmit_request <-> COM Outputs/Ctrl/Transmit request
//     PlcTask Outputs/GVL_iXlinker.Device_1_EtherCAT.Term_1_EK1200.Term_7_EL6001.COM_Outputs.Data_Out[{0..21}] <-> COM Outputs/Data Out {0..21}  (22 links)
//   TcoIoTests/TcoIoTests Instance <-> Device 4 (EtherCAT)
//     PlcTask Inputs/GVL_iXlinker.Device_4_EtherCAT.InfoData.AmsNetId <-> InfoData/AmsNetId
//     PlcTask Inputs/GVL_iXlinker.Device_4_EtherCAT.InfoData.CfgSlaveCount <-> InfoData/CfgSlaveCount
//     PlcTask Inputs/GVL_iXlinker.Device_4_EtherCAT.InfoData.ChangeCount <-> InfoData/ChangeCount
//     PlcTask Inputs/GVL_iXlinker.Device_4_EtherCAT.InfoData.DevId <-> InfoData/DevId
//     PlcTask Inputs/GVL_iXlinker.Device_4_EtherCAT.Inputs.DevState <-> Inputs/DevState
//     PlcTask Inputs/GVL_iXlinker.Device_4_EtherCAT.Inputs.Frm0InputToggle <-> Inputs/Frm0InputToggle
//     PlcTask Inputs/GVL_iXlinker.Device_4_EtherCAT.Inputs.Frm0State <-> Inputs/Frm0State
//     PlcTask Inputs/GVL_iXlinker.Device_4_EtherCAT.Inputs.Frm0WcState <-> Inputs/Frm0WcState
//     PlcTask Inputs/GVL_iXlinker.Device_4_EtherCAT.Inputs.SlaveCount <-> Inputs/SlaveCount
//     PlcTask Outputs/GVL_iXlinker.Device_4_EtherCAT.Outputs.DevCtrl <-> Outputs/DevCtrl
//     PlcTask Outputs/GVL_iXlinker.Device_4_EtherCAT.Outputs.Frm0Ctrl <-> Outputs/Frm0Ctrl
//     PlcTask Outputs/GVL_iXlinker.Device_4_EtherCAT.Outputs.Frm0WcCtrl <-> Outputs/Frm0WcCtrl
//   TcoIoTests/TcoIoTests Instance <-> Device 4 (EtherCAT)/Term 9 (EK1100)
//     PlcTask Inputs/GVL_iXlinker.Device_4_EtherCAT.Term_9_EK1100.InfoData.State <-> InfoData/State

CONFIGURATION TcoIo
    RESOURCE PLC ON TwinCAT3
        TASK PlcTask(INTERVAL := T#15ms, PRIORITY := 12);
        PROGRAM MAIN WITH PlcTask : MAIN;
    END_RESOURCE
END_CONFIGURATION

// ---- Diagnostics/EtherCAT/MasterDevice/Base/EtcMasterBase_62654B43.TcDUT
TYPE EtcMasterBase_62654B43 :
STRUCT
END_STRUCT
END_TYPE

// ---- Diagnostics/EtherCAT/MasterDevice/Base/SyncUnitsBase_AD6C35CE.TcDUT
TYPE SyncUnitsBase_AD6C35CE :
STRUCT
END_STRUCT
END_TYPE

// ---- Diagnostics/EtherCAT/MasterDevice/Base/SyncUnitTaskBase_FCD3CBF3.TcDUT
TYPE SyncUnitTaskBase_FCD3CBF3 :
STRUCT
END_STRUCT
END_TYPE

// ---- Diagnostics/EtherCAT/MasterDevice/Base/SyncUnitTasksBase_7C8711EB.TcDUT
TYPE SyncUnitTasksBase_7C8711EB :
STRUCT
END_STRUCT
END_TYPE

// ---- Diagnostics/EtherCAT/MasterDevice/SyncUnit/InfoData_8649EEEB.TcDUT
{attribute 'GeneratedUsingTerminal: IODEVICETYPE_ETHERCATPROT'}
{attribute addProperty BoxType "IODEVICETYPE_ETHERCATPROT"}
{attribute addProperty Id "ObjectIdAT %I*DWORD4StateAT %I*UINT2SlaveCountAT %I*UINT2"}
{attribute addProperty CRC "2252992235"}
{attribute addProperty Size "8"}
TYPE InfoData_8649EEEB :
STRUCT
    {attribute addProperty Name "ObjectId"}
    ObjectId AT %I* : DWORD;
    {attribute addProperty Name "State"}
    State AT %I* : UINT;
    {attribute addProperty Name "SlaveCount"}
    SlaveCount AT %I* : UINT;
END_STRUCT
END_TYPE

// ---- Diagnostics/EtherCAT/MasterDevice/SyncUnit/SyncUnitState.TcDUT
TYPE SyncUnitState : 
STRUCT
    {attribute addProperty Name "At least one slave in 'INIT' state"}
    AtLeastOneSlaveInInitState : BOOL;
    {attribute addProperty Name "At least one slave in 'PREOP' state"}
    AtLeastOneSlaveInPreopState : BOOL;
    {attribute addProperty Name "At least one slave in 'BOOT' state"}
    AtLeastOneSlaveInBootState : BOOL;
    {attribute addProperty Name "At least one slave in 'SAFEOP' state"}
    AtLeastOneSlaveInSafeOpState : BOOL;
    {attribute addProperty Name "At least one slave in 'OP' state"}
    AtLeastOneSlaveInOpState : BOOL;
    {attribute addProperty Name "At least one slave signals error"}
    AtLeastOneSlaveSignalsError : BOOL;
    {attribute addProperty Name "Invalid vendorId, productCode... read"}
    InvalidVendoridOrProductcodeRead : BOOL;
    {attribute addProperty Name "Initialization error occurred"}
    InitializationErrorOccurred : BOOL;
    {attribute addProperty Name "At least one slave disabled"}
    AtLeastOneSlaveDisabled : BOOL;
    {attribute addProperty Name "At least one slave not present"}
    AtLeastOneSlaveNotPresent : BOOL;
    {attribute addProperty Name "At least one slave signals link error"}
    AtLeastOneSlaveSignalsLinkError : BOOL;
    {attribute addProperty Name "At least one slave signals missing link"}
    AtLeastOneSlaveSignalsMissingLink : BOOL;
    {attribute addProperty Name "At least one slave signals unexpected link"}
    AtLeastOneSlaveSignalsUnexpectedLink : BOOL;
END_STRUCT
END_TYPE

// ---- Diagnostics/EtherCAT/MasterDevice/SyncUnit/SyncUnitTask_AB2F5079.TcDUT
{attribute 'GeneratedUsingTerminal: IODEVICETYPE_ETHERCATPROT'}
{attribute addProperty BoxType "IODEVICETYPE_ETHERCATPROT"}
{attribute addProperty Id "WcStateAT %I*WcState_0B2B16F91InfoDataAT %I*InfoData_8649EEEB8"}
{attribute addProperty CRC "2872004729"}
{attribute addProperty Size "9"}
TYPE SyncUnitTask_AB2F5079 EXTENDS SyncUnitTaskBase_FCD3CBF3 :
STRUCT
    {attribute addProperty Name "WcState"}
    WcState : WcState_0B2B16F9;
    {attribute addProperty Name "InfoData"}
    InfoData : InfoData_8649EEEB;
END_STRUCT
END_TYPE

// ---- Diagnostics/EtherCAT/SlaveDevice/Base/EtcSlaveBase_82538BE2.TcDUT
TYPE EtcSlaveBase_82538BE2 :
STRUCT
END_STRUCT
END_TYPE

// ---- Diagnostics/EtherCAT/SlaveDevice/Base/EtcSlaveBoxBase_77A0E4A7.TcDUT
{attribute clr[Container(Layout.Stack)]}
{attribute clr[Group(Layout.GroupBox)]}
{attribute addProperty PreviousPort "Unknown"}
{attribute addProperty SyncUnit "Unknown"}
TYPE EtcSlaveBoxBase_77A0E4A7 EXTENDS EtcSlaveBase_82538BE2 :
STRUCT
END_STRUCT
END_TYPE

// ---- Diagnostics/EtherCAT/SlaveDevice/Base/EtcSlaveEndTerminalBase_866C7F0C.TcDUT
{attribute clr[Container(Layout.Stack)]}
{attribute clr[Group(Layout.GroupBox)]}
{attribute addProperty PreviousPort "Unknown"}
{attribute addProperty SyncUnit "Unknown"}
TYPE EtcSlaveEndTerminalBase_866C7F0C EXTENDS EtcSlaveBase_82538BE2 :
STRUCT
END_STRUCT
END_TYPE

// ---- Diagnostics/EtherCAT/SlaveDevice/Base/EtcSlaveTerminalBase_947E5A46.TcDUT
{attribute clr[Container(Layout.Stack)]}
{attribute clr[Group(Layout.GroupBox)]}
{attribute addProperty PreviousPort "Unknown"}
{attribute addProperty SyncUnit "Unknown"}
TYPE EtcSlaveTerminalBase_947E5A46 EXTENDS EtcSlaveBase_82538BE2 :
STRUCT
END_STRUCT
END_TYPE

// ---- Diagnostics/EtherCAT/MasterDevice/InfoData_84133AC9.TcDUT
{attribute 'GeneratedUsingTerminal: IODEVICETYPE_ETHERCATPROT'}
{attribute addProperty BoxType "IODEVICETYPE_ETHERCATPROT"}
{attribute addProperty Id "ChangeCountAT %I*UINT2DevIdAT %I*UINT2AmsNetIdAT %I*AMSNETID6CfgSlaveCountAT %I*UINT2DcToTcTimeOffsetAT %I*LINT8DcToExtTimeOffsetAT %I*LINT8"}
{attribute addProperty CRC "3867959757"}
{attribute addProperty Size "28"}
TYPE InfoData_84133AC9 :
STRUCT
    {attribute addProperty Name "ChangeCount"}
    ChangeCount AT %I* : UINT;
    {attribute addProperty Name "DevId"}
    DevId AT %I* : UINT;
    {attribute addProperty Name "AmsNetId"}
    AmsNetId AT %I* : TcoAmsNetId;
    {attribute addProperty Name "CfgSlaveCount"}
    CfgSlaveCount AT %I* : UINT;
    {attribute addProperty Name "DcToTcTimeOffset"}
    DcToTcTimeOffset AT %I* : LINT;
    {attribute addProperty Name "DcToExtTimeOffset"}
    DcToExtTimeOffset AT %I* : LINT;
END_STRUCT
END_TYPE

// ---- Diagnostics/EtherCAT/MasterDevice/Inputs_A65FACA4.TcDUT
{attribute 'GeneratedUsingTerminal: IODEVICETYPE_ETHERCATPROT'}
{attribute addProperty BoxType "IODEVICETYPE_ETHERCATPROT"}
{attribute addProperty Id "SlaveCountAT %I*UINT2DevStateAT %I*UINT2Frm0StateAT %I*UINT2Frm0WcStateAT %I*UINT2Frm0InputToggleAT %I*UINT2"}
{attribute addProperty CRC "2791287972"}
{attribute addProperty Size "10"}
TYPE Inputs_A65FACA4 :
STRUCT
    {attribute addProperty Name "SlaveCount"}
    SlaveCount AT %I* : UINT;
    {attribute addProperty Name "DevState"}
    DevState AT %I* : UINT;
    {attribute addProperty Name "Frm0State"}
    Frm0State AT %I* : UINT;
    {attribute addProperty Name "Frm0WcState"}
    Frm0WcState AT %I* : UINT;
    {attribute addProperty Name "Frm0InputToggle"}
    Frm0InputToggle AT %I* : UINT;
END_STRUCT
END_TYPE

// ---- Diagnostics/EtherCAT/MasterDevice/Outputs_23C0ED1D.TcDUT
{attribute 'GeneratedUsingTerminal: IODEVICETYPE_ETHERCATPROT'}
{attribute addProperty BoxType "IODEVICETYPE_ETHERCATPROT"}
{attribute addProperty Id "DevCtrlAT %Q*UINT2Frm0CtrlAT %Q*UINT2Frm0WcCtrlAT %Q*UINT2"}
{attribute addProperty CRC "599846173"}
{attribute addProperty Size "6"}
TYPE Outputs_23C0ED1D :
STRUCT
    {attribute addProperty Name "DevCtrl"}
    DevCtrl AT %Q* : UINT;
    {attribute addProperty Name "Frm0Ctrl"}
    Frm0Ctrl AT %Q* : UINT;
    {attribute addProperty Name "Frm0WcCtrl"}
    Frm0WcCtrl AT %Q* : UINT;
END_STRUCT
END_TYPE

// ---- Diagnostics/EtherCAT/MasterDevice/TcoEthercatMasterDeviceState.TcDUT
TYPE TcoEthercatMasterDeviceState :
STRUCT
    {attribute addProperty Name "Link error"}
    LinkError : BOOL;
    {attribute addProperty Name "I/O locked after link error (I/O reset required)"}
    IOLockedAfterLinkError : BOOL;
    {attribute addProperty Name "Link error (redundancy adapter)"}
    LinkErrorRedundancyAdapter : BOOL;
    {attribute addProperty Name "Missing one frame (redundancy mode)"}
    MissingOneFrame : BOOL;
    {attribute addProperty Name "Out of send resources (I/O reset required)"}
    OutOfSendResources : BOOL;
    {attribute addProperty Name "Watchdog triggered"}
    WatchdogTriggered : BOOL;
    {attribute addProperty Name "Ethernet driver (miniport) not found"}
    EthernetDriverNotFound : BOOL;
    {attribute addProperty Name "I/O reset active"}
    IOResetActive : BOOL;
    {attribute addProperty Name "At least one slave in 'INIT' state"}
    AtLeastOneDeviceInInitState : BOOL;
    {attribute addProperty Name "At least one slave in 'PREOP' state"}
    AtLeastOneDeviceInPreOpState : BOOL;
    {attribute addProperty Name "At least one slave in 'SAFEOP' state"}
    AtLeastOneDeviceInSafeOpState : BOOL;
    {attribute addProperty Name "At least one device indicates an error state"}
    AtLeastOneDeviceIndicatesAnErrorState : BOOL;
    {attribute addProperty Name "DC not in sync"}
    DcNotInSync : BOOL;
END_STRUCT
END_TYPE

// ---- Diagnostics/EtherCAT/SlaveDevice/InfoData/InfoData_23CBA837.TcDUT
{attribute 'GeneratedUsingTerminal: EL6002-0000-0019'}
{attribute addProperty BoxType "EL6002-0000-0019"}
{attribute addProperty Id "AdsAddrAT %I*TcoIo.TcoAmsAddr0StateAT %I*UINT2"}
{attribute addProperty CRC "600549431"}
{attribute addProperty Size "2"}
TYPE InfoData_23CBA837 :
STRUCT
    {attribute addProperty Name "AdsAddr"}
    AdsAddr AT %I* : TcoAmsAddr;
    {attribute addProperty Name "State"}
    State AT %I* : UINT;
END_STRUCT
END_TYPE

// ---- Diagnostics/EtherCAT/SlaveDevice/InfoData/InfoData_6F19DB2B.TcDUT
{attribute 'GeneratedUsingTerminal: EL1809-0000-0018'}
{attribute addProperty BoxType "EL1809-0000-0018"}
{attribute addProperty Id "StateAT %I*UINT2"}
{attribute addProperty CRC "1863965483"}
{attribute addProperty Size "2"}
TYPE InfoData_6F19DB2B :
STRUCT
    {attribute addProperty Name "State"}
    State AT %I* : UINT;
END_STRUCT
END_TYPE

// ---- Diagnostics/EtherCAT/SlaveDevice/Inputs/InputBase_8311D824.TcDUT
TYPE InputBase_8311D824 :
STRUCT
END_STRUCT
END_TYPE

// ---- Diagnostics/EtherCAT/SlaveDevice/Outputs/OutputBase_10CEE7DE.TcDUT
TYPE OutputBase_10CEE7DE :
STRUCT
END_STRUCT
END_TYPE

// ---- Diagnostics/EtherCAT/SlaveDevice/WcState/WcState_0B2B16F9.TcDUT
{attribute 'GeneratedUsingTerminal: EL2809-0000-0018'}
{attribute addProperty BoxType "EL2809-0000-0018"}
{attribute addProperty Id "WcStateAT %I*BOOL1"}
{attribute addProperty CRC "187373305"}
{attribute addProperty Size "1"}
TYPE WcState_0B2B16F9 :
STRUCT
    {attribute addProperty Name "WcState"}
    WcState AT %I* : BOOL;
END_STRUCT
END_TYPE

// ---- Diagnostics/EtherCAT/SlaveDevice/WcState/WcState_9091E0EB.TcDUT
{attribute 'GeneratedUsingTerminal: EL6002-0000-0019'}
{attribute addProperty BoxType "EL6002-0000-0019"}
{attribute addProperty Id "WcStateAT %I*BOOL1InputToggleAT %I*BOOL1"}
{attribute addProperty CRC "2425479403"}
{attribute addProperty Size "2"}
TYPE WcState_9091E0EB :
STRUCT
    {attribute addProperty Name "WcState"}
    WcState AT %I* : BOOL;
    {attribute addProperty Name "InputToggle"}
    InputToggle AT %I* : BOOL;
END_STRUCT
END_TYPE

// ---- EtherCAT/eEcatState.TcDUT
{attribute 'qualified_only'}
TYPE eEcatState :
(
    MASK := 15,
    INIT := 1,
    PREOP := 2,
    BOOTSTRAP := 3,
    SAFEOP := 4,
    OP := 8,
    ERROR := 16,
    INVALID_VPRS := 32,
    INITCMD_ERROR := 48,
    DISABLED := 128
) BYTE;
END_TYPE

// ---- EtherCAT/eLinkState.TcDUT
{attribute 'qualified_only'}
TYPE eLinkState :
(
    EC_LINK_STATE_OK := 0,
    EC_LINK_STATE_NOT_PRESENT := 1,
    EC_LINK_STATE_LINK_WITHOUT_COMM := 2,
    EC_LINK_STATE_MISSING_LINK := 4,
    EC_LINK_STATE_ADDITIONAL_LINK := 8,
    EC_LINK_STATE_PORT_A := 16,
    EC_LINK_STATE_PORT_B := 32,
    EC_LINK_STATE_PORT_C := 64,
    EC_LINK_STATE_PORT_D := 128
) BYTE;
END_TYPE

// ---- SpecialPlcTypes/TcoAmsAddr.TcDUT
TYPE TcoAmsAddr :
STRUCT
    netId : ARRAY[0..5] OF BYTE;
    port : WORD;
END_STRUCT
END_TYPE

// ---- SpecialPlcTypes/TcoAmsNetId.TcDUT
TYPE TcoAmsNetId :
STRUCT
    netId : ARRAY[0..5] OF BYTE;
END_STRUCT
END_TYPE

// ---- Diagnostics/EtherCAT/TcoEthercat.TcGVL
{attribute 'qualified_only'}
VAR_GLOBAL CONSTANT
    C_MaxSyncUnits : UINT := 10;
    C_MAX_LOCAL_ERROR_MESSAGES : UINT := 3;
END_VAR

// ---- Diagnostics/EtherCAT/MasterDevice/SyncUnit/ITcoSyncUnit.TcIO
INTERFACE ITcoSyncUnit

PROPERTY DataInvalid : BOOL
GET
END_GET
END_PROPERTY

PROPERTY DataValid : BOOL
GET
END_GET
END_PROPERTY

PROPERTY HasSomeIssue : BOOL
GET
END_GET
END_PROPERTY

PROPERTY State : SyncUnitState
GET
END_GET
END_PROPERTY

END_INTERFACE

// ---- Diagnostics/EtherCAT/MasterDevice/ITcoEthercatMasterDevice.TcIO
INTERFACE ITcoEthercatMasterDevice

PROPERTY AllDataValid : BOOL
GET
END_GET
END_PROPERTY

PROPERTY DeviceHasSomeIssue : BOOL
GET
END_GET
END_PROPERTY

PROPERTY SomeDataInvalid : BOOL
GET
END_GET
END_PROPERTY

PROPERTY SomeSyncUnitHasSomeIssue : BOOL
GET
END_GET
END_PROPERTY

PROPERTY State : TcoEthercatMasterDeviceState
GET
END_GET
END_PROPERTY

END_INTERFACE

// ---- EtherCAT/ITcoEcatComponent.TcIO
INTERFACE ITcoEcatComponent

PROPERTY EcatState : REFERENCE TO TcoEcatSlaveState
GET
END_GET
END_PROPERTY

END_INTERFACE

// ---- POUs/MAIN.TcPOU
PROGRAM MAIN
VAR
END_VAR

END_PROGRAM

// ---- Diagnostics/EtherCAT/MasterDevice/SyncUnit/TcoSyncUnit.TcPOU
FUNCTION_BLOCK TcoSyncUnit EXTENDS TcoCore.TcoObject IMPLEMENTS ITcoSyncUnit
VAR
    {attribute addProperty Name "WcState"}
    WcState : WcState_0B2B16F9;
    {attribute addProperty Name "InfoData"}
    InfoData : InfoData_8649EEEB;
    {attribute addProperty Name "Status"}
    _State : SyncUnitState;
    {attribute 'hide'}
    _hasSomeIssue : BOOL;
    {attribute 'hide'}
    _dataValid : BOOL;
    {attribute 'hide'}
    _dataInvalid : BOOL;
END_VAR

PROPERTY DataInvalid : BOOL
GET
_dataInvalid := WcState.WcState;
DataInvalid := _dataInvalid;
END_GET
END_PROPERTY

PROPERTY DataValid : BOOL
GET
_dataValid := NOT WcState.WcState;
DataValid := _dataValid;
END_GET
END_PROPERTY

PROPERTY HasSomeIssue : BOOL
GET
VAR
    _syncUnitStatus : SyncUnitState;
END_VAR
_syncUnitStatus := State;

_hasSomeIssue := _syncUnitStatus.AtLeastOneSlaveInInitState OR
    _syncUnitStatus.AtLeastOneSlaveInPreopState OR
    _syncUnitStatus.AtLeastOneSlaveInBootState OR
    _syncUnitStatus.AtLeastOneSlaveInSafeOpState OR
    _syncUnitStatus.AtLeastOneSlaveSignalsError OR
    _syncUnitStatus.InvalidVendoridOrProductcodeRead OR
    _syncUnitStatus.InitializationErrorOccurred OR
    _syncUnitStatus.AtLeastOneSlaveNotPresent OR
    _syncUnitStatus.AtLeastOneSlaveSignalsLinkError OR
    _syncUnitStatus.AtLeastOneSlaveSignalsMissingLink OR
    _syncUnitStatus.AtLeastOneSlaveSignalsUnexpectedLink;

HasSomeIssue := _hasSomeIssue;
END_GET
END_PROPERTY

PROPERTY State : SyncUnitState
GET
_State.AtLeastOneSlaveInInitState := InfoData.State.0 AND NOT InfoData.State.1;
_State.AtLeastOneSlaveInPreopState := InfoData.State.0 AND InfoData.State.1;
_State.AtLeastOneSlaveInBootState := InfoData.State.0 AND InfoData.State.1;
_State.AtLeastOneSlaveInSafeOpState := InfoData.State.2;
_State.AtLeastOneSlaveInOpState := InfoData.State.3;
_State.AtLeastOneSlaveSignalsError := InfoData.State.4;
_State.InvalidVendoridOrProductcodeRead := InfoData.State.5;
_State.InitializationErrorOccurred := InfoData.State.6;
_State.AtLeastOneSlaveDisabled := InfoData.State.7;
_State.AtLeastOneSlaveNotPresent := InfoData.State.8;
_State.AtLeastOneSlaveSignalsLinkError := InfoData.State.9;
_State.AtLeastOneSlaveSignalsMissingLink := InfoData.State.10;
_State.AtLeastOneSlaveSignalsUnexpectedLink := InfoData.State.11;
State := _State;
END_GET
END_PROPERTY

END_FUNCTION_BLOCK

// ---- Diagnostics/EtherCAT/MasterDevice/Messenger/DiagnosticsMessenger.TcPOU
FUNCTION_BLOCK DiagnosticsMessenger EXTENDS TcoCore.TcoMessenger

{attribute 'hide'}
METHOD FB_init : BOOL
VAR_INPUT
    bInitRetains : BOOL; // if TRUE, the retain variables are initialized (warm start / cold start)
    bInCopyCode : BOOL; // if TRUE, the instance afterwards gets moved into the copy code (online change)
    ParentObject : ITcoObject;
END_VAR
END_METHOD

END_FUNCTION_BLOCK

// ---- Diagnostics/EtherCAT/MasterDevice/Messenger/DiagnosticsMessengers.TcPOU
FUNCTION_BLOCK DiagnosticsMessengers EXTENDS TcoCore.TcoObject
VAR
    Messengers : ARRAY[0..2] OF DiagnosticsMessenger(THIS^);
END_VAR

{attribute 'hide'}
METHOD FB_init : BOOL
VAR_INPUT
    bInitRetains : BOOL; // if TRUE, the retain variables are initialized (warm start / cold start)
    bInCopyCode : BOOL; // if TRUE, the instance afterwards gets moved into the copy code (online change)
    ParentObject : ITcoObject;
END_VAR
Messengers[0].FB_init(bInitRetains, bInCopyCode, ParentObject);
Messengers[1].FB_init(bInitRetains, bInCopyCode, ParentObject);
Messengers[2].FB_init(bInitRetains, bInCopyCode, ParentObject);
END_METHOD

END_FUNCTION_BLOCK

// ---- Diagnostics/EtherCAT/MasterDevice/TcoEthercatDiagnosticsTask.TcPOU
FUNCTION_BLOCK TcoEthercatDiagnosticsTask EXTENDS TcoCore.TcoTask
VAR_INPUT
    inNetId : Tc2_System.T_AmsNetID;
END_VAR
VAR
    _EcGetAllSlaveStates : Tc2_EtherCAT.FB_EcGetAllSlaveStates;
    _EcGetConfSlaves : Tc2_EtherCAT.FB_EcGetConfSlaves;
    _updateDiagnosticsState : TcoCore.TcoState(THIS^, TcoCore.eRestoreMode.None);
    _SlaveStatesCount : UINT;
    _ConfigSlavesCount : UINT;
    _SlaveStateBuffer : ARRAY[0..EC_MAX_SLAVES] OF Tc2_EtherCAT.ST_EcSlaveState;
    _SlaveConfigDataBuffer : ARRAY[0..EC_MAX_SLAVES] OF Tc2_EtherCAT.ST_EcSlaveConfigData;
    _i : UINT;
    _name : STRING;
    _type : STRING;
    _state : STRING;
    _DiagnosticsMessengers : DiagnosticsMessengers(THIS^);
    _DiagnosticsMessengerIndex : UINT;
END_VAR
VAR_OUTPUT
    outDiagnosticsAvailable : BOOL;
END_VAR

IF Execute() THEN
    IF _updateDiagnosticsState.State = 10 THEN
        outDiagnosticsAvailable := FALSE;
        _EcGetAllSlaveStates(bExecute := FALSE);
        _EcGetConfSlaves(bExecute := FALSE);

        IF NOT _EcGetAllSlaveStates.bBusy AND NOT _EcGetAllSlaveStates.bError AND NOT _EcGetConfSlaves.bBusy AND NOT _EcGetConfSlaves.bError THEN
            _updateDiagnosticsState.ChangeState(_updateDiagnosticsState._State + 10);
        END_IF
    END_IF

    IF _updateDiagnosticsState.State = 20 THEN
        _EcGetAllSlaveStates(sNetId := inNetId,
            pStateBuf := ADR(_SlaveStateBuffer),
            cbBufLen := SIZEOF(_SlaveStateBuffer),
            bExecute := TRUE,
            tTimeout :=,
            bBusy =>,
            bError =>,
            nErrId =>,
            nSlaves => _SlaveStatesCount);

        IF _EcGetAllSlaveStates.bBusy THEN
            _updateDiagnosticsState.ChangeState(_updateDiagnosticsState._State + 10);
        END_IF
    END_IF

    IF _updateDiagnosticsState.State = 30 THEN
        _EcGetAllSlaveStates(sNetId := inNetId,
            pStateBuf := ADR(_SlaveStateBuffer),
            cbBufLen := SIZEOF(_SlaveStateBuffer),
            bExecute := FALSE,
            tTimeout :=,
            bBusy =>,
            bError =>,
            nErrId =>,
            nSlaves => _SlaveStatesCount);

        IF NOT _EcGetAllSlaveStates.bBusy AND NOT _EcGetAllSlaveStates.bError THEN
            _updateDiagnosticsState.ChangeState(_updateDiagnosticsState._State + 10);
        END_IF
    END_IF

    IF _updateDiagnosticsState.State = 40 THEN
        _EcGetConfSlaves(sNetId := inNetId,
            pArrEcConfSlaveInfo := ADR(_SlaveConfigDataBuffer),
            cbBufLen := SIZEOF(_SlaveConfigDataBuffer),
            bExecute := TRUE,
            tTimeout :=,
            bBusy =>,
            bError =>,
            nErrorId =>,
            nSlaves => _ConfigSlavesCount);

        IF _EcGetConfSlaves.bBusy THEN
            _updateDiagnosticsState.ChangeState(_updateDiagnosticsState._State + 10);
        END_IF
    END_IF

    IF _updateDiagnosticsState.State = 50 THEN
        _EcGetConfSlaves(sNetId := inNetId,
            pArrEcConfSlaveInfo := ADR(_SlaveConfigDataBuffer),
            cbBufLen := SIZEOF(_SlaveConfigDataBuffer),
            bExecute := FALSE,
            tTimeout :=,
            bBusy =>,
            bError =>,
            nErrorId =>,
            nSlaves => _ConfigSlavesCount);

        IF NOT _EcGetConfSlaves.bBusy AND NOT _EcGetConfSlaves.bError THEN
            _updateDiagnosticsState.ChangeState(_updateDiagnosticsState._State + 10);
        END_IF
    END_IF

    IF _updateDiagnosticsState.State = 60 THEN
        _EcGetAllSlaveStates(bExecute := FALSE);
        _EcGetConfSlaves(bExecute := FALSE);

        IF NOT _EcGetAllSlaveStates.bBusy AND NOT _EcGetAllSlaveStates.bError AND NOT _EcGetConfSlaves.bBusy AND NOT _EcGetConfSlaves.bError THEN
            _updateDiagnosticsState.ChangeState(_updateDiagnosticsState._State + 10);
        END_IF
    END_IF

    IF _updateDiagnosticsState.State = 70 THEN
        _DiagnosticsMessengerIndex := 0;

        FOR _i := 0 TO _ConfigSlavesCount DO
            IF (_SlaveStateBuffer[_i].deviceState <> 8 OR _SlaveStateBuffer[_i].linkState <> 0) THEN
                IF _SlaveConfigDataBuffer[_i].sName <> '' THEN
                    IF _DiagnosticsMessengerIndex <= 2 THEN
                        outDiagnosticsAvailable := TRUE;
                        _name := _SlaveConfigDataBuffer[_i].sName;
                        _type := Tc2_EtherCAT.F_ConvProductCodeToString(_SlaveConfigDataBuffer[_i].stSlaveIdentity);
                        _state := Tc2_EtherCAT.F_ConvSlaveStateToString(state := _SlaveStateBuffer[_i]);

                        _DiagnosticsMessengers.Messengers[_DiagnosticsMessengerIndex].Build()
                            .AppendAny(_name)
                            .Append('[')
                            .AppendAny(_type)
                            .Append(']')
                            .Append(_state)
                            .As()
                            .AsError().Pin();

                        _DiagnosticsMessengerIndex := _DiagnosticsMessengerIndex + 1;
                    END_IF
                END_IF
            END_IF;
        END_FOR

        _updateDiagnosticsState.ChangeState(_updateDiagnosticsState._State + 10);
    END_IF

    IF _updateDiagnosticsState.State = 80 THEN
        DoneWhen(TRUE);
    END_IF

    ThrowWhen(_EcGetAllSlaveStates.bError OR _EcGetConfSlaves.bError);
END_IF

METHOD FB_init : BOOL
VAR_INPUT
    bInitRetains : BOOL; // if TRUE, the retain variables are initialized (warm start / cold start)
    bInCopyCode : BOOL; // if TRUE, the instance afterwards gets moved into the copy code (online change)
    ParentObject : TcoCore.ITcoObject;
END_VAR
END_METHOD

(*~
    <docu>
        <summary>
            Executes when task is aborted.
        </summary>
    </docu>
~*)
METHOD PROTECTED OnAbort
_EcGetAllSlaveStates(bExecute := FALSE);
_EcGetConfSlaves(bExecute := FALSE);
_updateDiagnosticsState.Restore();
END_METHOD

(*~
    <docu>
        <summary>
            Executes when task reaches the ```Done``` state .
        </summary>
    </docu>
~*)
METHOD PROTECTED OnDone
_EcGetAllSlaveStates(bExecute := FALSE);
_EcGetConfSlaves(bExecute := FALSE);
END_METHOD

(*~
    <docu>
        <summary>
            Executes when task reaches the ```Error``` state.
            <para>
                Do not confuse with <see cref="PlcDocu.TcoCore.TcoTask.WhileError()"/>, that is called cyclically until '''Error''' state is left.
            </para>
        </summary>
    </docu>
~*)
METHOD PROTECTED OnError
IF _EcGetAllSlaveStates.bError THEN
    Messenger.Build()
        .Append('Reading status of all EtherCAT slaves using "Tc2_EtherCAT.FB_EcGetAllSlaveStates" function block returns error. nErrId: ')
        .AppendAny(_EcGetAllSlaveStates.nErrId)
        .As().AsError();
ELSIF _EcGetConfSlaves.bError THEN
    Messenger.Build()
        .Append('Reading status of configurateed EtherCAT slaves using "Tc2_EtherCAT.FB_EcGetConfSlaves" function block returns error. nErrorId: ')
        .AppendAny(_EcGetConfSlaves.nErrorId)
        .As().AsError();
END_IF
END_METHOD

METHOD PROTECTED OnStart
_EcGetAllSlaveStates(bExecute := FALSE);
_EcGetConfSlaves(bExecute := FALSE);
_updateDiagnosticsState.ChangeState(10);
END_METHOD

(*~
    <docu>
        <summary>
            Restores this instance to the Ready state. Can be called explicitly or from within one of the restore mechanisms.
            <para>
                See also <see cref="PlcDocu.TcoCore.TcoTask.AutoRestorable()"/>
            </para>
        </summary>
    </docu>
~*)
METHOD Restore : ITcoRestorable
THIS^._EcGetAllSlaveStates(bExecute := FALSE);
THIS^._EcGetConfSlaves(bExecute := FALSE);
THIS^._DiagnosticsMessengers.Messengers[0].Clear();
THIS^._DiagnosticsMessengers.Messengers[1].Clear();
THIS^._DiagnosticsMessengers.Messengers[2].Clear();
THIS^.outDiagnosticsAvailable := FALSE;
THIS^._updateDiagnosticsState.Restore();
SUPER^.Restore();
END_METHOD

END_FUNCTION_BLOCK

// ---- Diagnostics/EtherCAT/MasterDevice/TcoEthercatMasterDevice.TcPOU
FUNCTION_BLOCK TcoEthercatMasterDevice EXTENDS TcoCore.TcoComponent IMPLEMENTS ITcoEthercatMasterDevice
VAR_INPUT
    Inputs : Inputs_A65FACA4;
    InfoData : InfoData_84133AC9;
    SyncUnits : POINTER TO SyncUnitTask_AB2F5079;
    SyncUnitsSize : UINT;
END_VAR
VAR
    _someSyncUnitHasSomeIssue : BOOL;
    _allDataValid : BOOL;
    _someDataInvalid : BOOL;
    _State : TcoEthercatMasterDeviceState;
    _NetId : Tc2_System.T_AmsNetID;
    _DeviceHasSomeIssue : BOOL;
    _TcoEthercatDiagnosticsTask : TcoEthercatDiagnosticsTask(THIS^);
    _InfoDataChangeCountPV : UINT;
    _numberOfSyncUnits : UINT;
    {attribute addProperty Name "Acknowledge"}
    _acknowledge : TcoCore.TcoTask(THIS^);
    _DiagnosticsAvailable : BOOL;
END_VAR
VAR_OUTPUT
    Outputs : Outputs_23C0ED1D;
END_VAR

UpdateSyncUnitsStatus(SyncUnits, SyncUnitsSize);
Diagnostics();

PROPERTY AllDataValid : BOOL
GET
AllDataValid := _allDataValid;
END_GET
END_PROPERTY

PROPERTY DeviceHasSomeIssue : BOOL
GET
_DeviceHasSomeIssue := _State.LinkError OR
    _State.IOLockedAfterLinkError OR
    _State.LinkErrorRedundancyAdapter OR
    _State.MissingOneFrame OR
    _State.OutOfSendResources OR
    _State.WatchdogTriggered OR
    _State.EthernetDriverNotFound OR
    _State.IOResetActive OR
    _State.AtLeastOneDeviceInInitState OR
    _State.AtLeastOneDeviceInPreOpState OR
    _State.AtLeastOneDeviceInSafeOpState OR
    _State.AtLeastOneDeviceIndicatesAnErrorState OR
    _State.DcNotInSync;

DeviceHasSomeIssue := _DeviceHasSomeIssue;
END_GET
END_PROPERTY

METHOD Diagnostics
VAR
    _i : UINT;
END_VAR
_NetId := Tc2_System.F_CreateAmsNetId(InfoData.AmsNetId.netId);
_TcoEthercatDiagnosticsTask(inNetId := _NetId, outDiagnosticsAvailable => _DiagnosticsAvailable);
Service();

IF _acknowledge.Execute() THEN
    Restore();
END_IF

IF (DeviceHasSomeIssue OR SomeSyncUnitHasSomeIssue OR SomeDataInvalid OR _InfoDataChangeCountPV <> InfoData.ChangeCount
    ) (*OR _manualDiagnosticStart.Execute()*) THEN
    IF _TcoEthercatDiagnosticsTask.Ready THEN
        _InfoDataChangeCountPV := InfoData.ChangeCount;
        _TcoEthercatDiagnosticsTask.Invoke();
    END_IF

    IF _TcoEthercatDiagnosticsTask.Done AND NOT _DiagnosticsAvailable THEN
        _TcoEthercatDiagnosticsTask.Restore();
    END_IF;
END_IF
END_METHOD

METHOD FB_init : BOOL
VAR_INPUT
    bInitRetains : BOOL; // if TRUE, the retain variables are initialized (warm start / cold start)
    bInCopyCode : BOOL; // if TRUE, the instance afterwards gets moved into the copy code (online change)
    ParentObject : TcoCore.ITcoObject;
END_VAR
END_METHOD

(*~
    <docu>
        <summary>
            Restores this instance to the Ready state. Can be called explicitly or from within one of the restore mechanisms.
        </summary>
    </docu>
~*)
METHOD Restore : ITcoRestorable
THIS^.Messenger.Clear();
THIS^._DiagnosticsAvailable := FALSE;
THIS^._acknowledge.Restore();
THIS^._TcoEthercatDiagnosticsTask.Restore();
END_METHOD

(*~
    <docu>
        <summary>
            Custom service (manual, maintenance) logic.
            This method must be implemented in derived class.
        </summary>
    </docu>
~*)
METHOD PROTECTED ServiceMode
_acknowledge();
END_METHOD

PROPERTY SomeDataInvalid : BOOL
GET
SomeDataInvalid := _someDataInvalid;
END_GET
END_PROPERTY

PROPERTY SomeSyncUnitHasSomeIssue : BOOL
GET
SomeSyncUnitHasSomeIssue := _someSyncUnitHasSomeIssue;
END_GET
END_PROPERTY

PROPERTY State : TcoEthercatMasterDeviceState
GET
_State.LinkError := Inputs.DevState.0;
_State.IOLockedAfterLinkError := Inputs.DevState.1;
_State.LinkErrorRedundancyAdapter := Inputs.DevState.2;
_State.MissingOneFrame := Inputs.DevState.3;
_State.OutOfSendResources := Inputs.DevState.4;
_State.WatchdogTriggered := Inputs.DevState.5;
_State.EthernetDriverNotFound := Inputs.DevState.6;
_State.IOResetActive := Inputs.DevState.7;
_State.AtLeastOneDeviceInInitState := Inputs.DevState.8;
_State.AtLeastOneDeviceInPreOpState := Inputs.DevState.9;
_State.AtLeastOneDeviceInSafeOpState := Inputs.DevState.10;
_State.AtLeastOneDeviceIndicatesAnErrorState := Inputs.DevState.11;
_State.DcNotInSync := Inputs.DevState.12;
State := _State;
END_GET
END_PROPERTY

METHOD SyncUnitHasSomeIssue : BOOL
VAR_INPUT
    inState : UINT;
END_VAR
VAR
    _state : SyncUnitState;
END_VAR
_state.AtLeastOneSlaveInInitState := inState.0 AND NOT inState.1;
_state.AtLeastOneSlaveInPreopState := inState.0 AND inState.1;
_state.AtLeastOneSlaveInBootState := inState.0 AND inState.1;
_state.AtLeastOneSlaveInSafeOpState := inState.2;
_state.AtLeastOneSlaveInOpState := inState.3;
_state.AtLeastOneSlaveSignalsError := inState.4;
_state.InvalidVendoridOrProductcodeRead := inState.5;
_state.InitializationErrorOccurred := inState.6;
_state.AtLeastOneSlaveDisabled := inState.7;
_state.AtLeastOneSlaveNotPresent := inState.8;
_state.AtLeastOneSlaveSignalsLinkError := inState.9;
_state.AtLeastOneSlaveSignalsMissingLink := inState.10;
_state.AtLeastOneSlaveSignalsUnexpectedLink := inState.11;

SyncUnitHasSomeIssue := _state.AtLeastOneSlaveInInitState OR
    _state.AtLeastOneSlaveInPreopState OR
    _state.AtLeastOneSlaveInBootState OR
    _state.AtLeastOneSlaveInSafeOpState OR
    _state.AtLeastOneSlaveSignalsError OR
    _state.InvalidVendoridOrProductcodeRead OR
    _state.InitializationErrorOccurred OR
    _state.AtLeastOneSlaveNotPresent OR
    _state.AtLeastOneSlaveSignalsLinkError OR
    _state.AtLeastOneSlaveSignalsMissingLink OR
    _state.AtLeastOneSlaveSignalsUnexpectedLink;
END_METHOD

METHOD UpdateSyncUnitsStatus
VAR_INPUT
    SyncUnits : POINTER TO SyncUnitTask_AB2F5079;
    SyncUnitsSize : UINT;
END_VAR
VAR
    _i : UINT;
    _pSyncUnit : POINTER TO SyncUnitTask_AB2F5079;
    _SyncUnit : SyncUnitTask_AB2F5079;
    _SyncUnitState : UINT;
END_VAR
_someSyncUnitHasSomeIssue := FALSE;
_allDataValid := TRUE;
_someDataInvalid := FALSE;

IF SyncUnits <> 0 THEN
    _numberOfSyncUnits := SyncUnitsSize / SIZEOF(SyncUnitTask_AB2F5079);

    FOR _i := 0 TO _numberOfSyncUnits - 1 DO
        _pSyncUnit := SyncUnits + _i * SIZEOF(SyncUnitTask_AB2F5079);
        _SyncUnit := _pSyncUnit^;
        _someSyncUnitHasSomeIssue := _someSyncUnitHasSomeIssue OR SyncUnitHasSomeIssue(_SyncUnit.InfoData.State);
        _allDataValid := _allDataValid AND NOT _SyncUnit.WcState.WcState;
        _someDataInvalid := _someDataInvalid OR _SyncUnit.WcState.WcState;
    END_FOR
END_IF
END_METHOD

END_FUNCTION_BLOCK

// ---- Diagnostics/ProfinetComponent/TcoPnIoComponent.TcPOU
FUNCTION_BLOCK ABSTRACT TcoPnIoComponent EXTENDS TcoCore.TcoComponent
VAR_INPUT
    inPnIoBoxState : UINT;
    inPnIoBoxDiag : UINT;
END_VAR
VAR
    //*{attribute addProperty Name "<#PN ready#>"}
    //*{attribute clr [ReadOnly()]}
    _profinetReady : BOOL;
END_VAR

//PnIoBoxState
//0 = No error
//1 = Profinet device state machine is in boot mode
//2 = Device not found
//3 = The stationname is not unique
//4 = IP could not be set
//5 = IP conflict
//6 = DCP set was not successful
//7 = Watchdog error
//8 = Datahold error
//9 = RTC3: Sync mode could not be initiated
//10 = Profinet controller has a link error
//11 = The aliasname is not unique
//12 = The automatic name assignement isn't possible - wrong device type
//13 = IOC-AR is established but no application ready
//14 = IOC-AR is established but module difference
//15 = At least one InputCR is invalid, provider in stop or problemindicator is set
//16 = At least one OutputCR is invalid, provider in stop or problemindicator is set
//31 = Only for EtherCAT gateways: WC-State of cyclic EtherCAT frame is 1
THIS^.Messenger.OnCondition(inPnIoBoxState = 1).Error('<#Profinet device state machine is in boot mode!#>');
THIS^.Messenger.OnCondition(inPnIoBoxState = 2).Error('<#Device NOT found!#>');
THIS^.Messenger.OnCondition(inPnIoBoxState = 3).Error('<#The stationname is not unique!#>');
THIS^.Messenger.OnCondition(inPnIoBoxState = 4).Error('<#IP could NOT be set!#>');
THIS^.Messenger.OnCondition(inPnIoBoxState = 5).Error('<#IP conflict!#>');
THIS^.Messenger.OnCondition(inPnIoBoxState = 6).Error('<#DCP set was NOT successful!#>');
THIS^.Messenger.OnCondition(inPnIoBoxState = 7).Error('<#Watchdog error!#>');
THIS^.Messenger.OnCondition(inPnIoBoxState = 8).Error('<#Datahold error!#>');
THIS^.Messenger.OnCondition(inPnIoBoxState = 9).Error('<#RTC3: Sync mode could not be initiated!#>');
THIS^.Messenger.OnCondition(inPnIoBoxState = 10).Error('<#Profinet controller has a link error!#>');
THIS^.Messenger.OnCondition(inPnIoBoxState = 11).Error('<#The aliasname is not unique!#>');
THIS^.Messenger.OnCondition(inPnIoBoxState = 12).Error('<#The automatic name assignement is not possible - wrong device TYPE!#>');
THIS^.Messenger.OnCondition(inPnIoBoxState = 13).Error('<#IOC-AR is established but no application ready!#>');
THIS^.Messenger.OnCondition(inPnIoBoxState = 14).Error('<#IOC-AR is established but module difference!#>');
THIS^.Messenger.OnCondition(inPnIoBoxState = 15).Error('<#AT least one InputCR is invalid, provider in stop OR problemindicator is set!#>');
THIS^.Messenger.OnCondition(inPnIoBoxState = 16).Error('<#At least one OutputCR is invalid, provider in stop or problemindicator is set!#>');
THIS^.Messenger.OnCondition(inPnIoBoxState = 31).Error('<#EtherCAT gateway: WC-State OF cyclic EtherCAT frame is 1!#>');
//PnIoBoxDiag
//0x0000 = No diagnosis
//0x0001 = IOC-AR is not established
//0x0002 = IOC-AR is established
//0x0004 = IOC-AR is established but no application ready
//0x0008 = IOC-AR is established but module difference
//0x0010 = At least one AlarmCR got a diagnosis alarm
//0x0100 = At least one InputCR is invalid
//0x0200 = At least one InputCR Provider is in stop
//0x0400 = At least one InputCR Problemindicator is set
//0x1000 = At least one OutputCR is invalid
//0x2000 = At least one OutputCR Provider is in stop
//0x4000 = At least one OutputCR Problemindicator is set
THIS^.Messenger.OnCondition(inPnIoBoxDiag.0).Error('<#IOC-AR is not established!#>');
THIS^.Messenger.OnCondition(NOT _profinetReady AND inPnIoBoxDiag.1).Info('<#IOC-AR is established!#>');
THIS^.Messenger.OnCondition(inPnIoBoxDiag.2).Error('<#IOC-AR is established but no application ready!#>');
THIS^.Messenger.OnCondition(inPnIoBoxDiag.3).Error('<#IOC-AR is established but module difference!#>');
THIS^.Messenger.OnCondition(inPnIoBoxDiag.4).Error('<#AT least one AlarmCR got a diagnosis alarm!#>');
THIS^.Messenger.OnCondition(inPnIoBoxDiag.8).Error('<#At least one InputCR is invalid!#>');
THIS^.Messenger.OnCondition(inPnIoBoxDiag.9).Error('<#AT least one InputCR Provider is in stop!#>');
THIS^.Messenger.OnCondition(inPnIoBoxDiag.10).Error('<#At least one InputCR Problemindicator is set!#>');
THIS^.Messenger.OnCondition(inPnIoBoxDiag.12).Error('<#AT least one OutputCR is invalid!#>');
THIS^.Messenger.OnCondition(inPnIoBoxDiag.13).Error('<#At least one OutputCR Provider is in stop!#>');
THIS^.Messenger.OnCondition(inPnIoBoxDiag.14).Error('<#AT least one OutputCR Problemindicator is set!#>');
_profinetReady := inPnIoBoxState = 0 AND inPnIoBoxDiag = 2;

PROPERTY ProfinetReady : BOOL
GET
ProfinetReady := _profinetReady;
END_GET
END_PROPERTY

END_FUNCTION_BLOCK

// ---- EtherCAT/TcoEcatSlaveState.TcPOU
FUNCTION_BLOCK TcoEcatSlaveState EXTENDS TcoObject
VAR_INPUT
    AdsAddr : AMSADDR;
END_VAR
VAR_OUTPUT
END_VAR
VAR
    //*	{attribute addProperty Name "<#Actual state#>"}
    //*	{attribute clr [ReadOnly()]}
    _ecatState : eEcatState;
    //*	{attribute addProperty Name "<#Actual Link state#>"}
    //*	{attribute clr [ReadOnly()]}
    _linkState : eLinkState;
    //*	{attribute addProperty Name "<#ECAT Communication Ok#>"}
    //*	{attribute clr [ReadOnly()]}
    _ecatOk : BOOL;
    //*	{attribute clr [RenderIgnore()]}
    _progress : INT := 0;
    //*	{attribute addProperty Name "<#EtherCat masters Ams Net Id#>"}
    //*	{attribute clr [ReadOnly()]}
    _netId : STRING[23]; //as string
    //* {attribute clr [RenderIgnore()]}
    _etherCAT_Addr : UINT;
    //*	{attribute addProperty Name "<#State check Time(Period)#>"}
    _periodStateCheckTime : TIME := T#1S;
    //*	{attribute addProperty Name "<#Error Time#>"}
    _errorTime : TIME := T#5S;
    //*	{attribute clr [RenderIgnore()]}
    _getSlaveState : FB_EcGetSlaveState;
    //*	{attribute clr [RenderIgnore()]}
    _setSlaveState : FB_EcSetSlaveState;
    //*	{attribute clr [RenderIgnore()]}
    bExecute : BOOL;
    //*	{attribute clr [RenderIgnore()]}
    state : ST_EcSlaveState;
    //*	{attribute clr [RenderIgnore()]}
    _error : BOOL;
    //*	{attribute clr [RenderIgnore()]}
    _busy : BOOL;
    //*	{attribute clr [RenderIgnore()]}
    _errId : UDINT;
    //*	{attribute clr [RenderIgnore()]}
    _stateTimer : TON;
    //*	{attribute clr [RenderIgnore()]}
    _errorTimer : TON;
    //*	{attribute addProperty Name "<#Required state#>"}
    _ecatReqestState : eEcatState;
    //*	{attribute addProperty Name "<#Change State#>"}
    _changeStateTask : TcoCore.TcoTask(THIS^);
    //*	{attribute addProperty Name "<#Restore#>"}
    _restoreTask : TcoCore.TcoTask(THIS^);
    {attribute 'hide'}
    _sb : TcoCore.StringBuilder;
    {attribute 'hide'}
    _amsEmpty : BOOL;
END_VAR

_netId := F_CreateAmsNetId(nIds := AdsAddr.netId);
_etherCAT_Addr := AdsAddr.port;
_amsEmpty := (_netId = '0.0.0.0.0.0') OR (_etherCAT_Addr = 0);

IF _changeStateTask.Execute() THEN
    _changeStateTask.DoneWhen(ChangeState(RequestedDeviceState := _ecatReqestState));
END_IF

THIS^._changeStateTask.ThrowWhen((_changeStateTask.ElapsedTime >= _errorTime AND _progress > 0) OR _amsEmpty);
THIS^._changeStateTask.Messenger.OnCondition(_amsEmpty).Error('<#Ads address information is not defined!#>');
//*************RESTORE********************
_restoreTask.Enabled := TRUE;

IF _restoreTask.Execute() THEN
    Restore();
END_IF

//****************************************
IF (_amsEmpty) THEN
    RETURN;
END_IF

THIS^._GetState(_periodStateCheckTime);

METHOD PRIVATE _GetState
VAR_INPUT
    Period : TIME;
END_VAR
_stateTimer(IN := TRUE, PT := Period);

IF _stateTimer.Q THEN
    bExecute := TRUE;
    _stateTimer(IN := FALSE);
END_IF

_getSlaveState(sNetId := _netId,
    nSlaveAddr := _etherCAT_Addr,
    bExecute := bExecute,
    bBusy => _busy,
    state => state,
    bError => _error,
    nErrId => _ErrId);

IF NOT _busy THEN
    _ecatState := state.deviceState;
    _linkState := state.linkState;
    _ecatOk := (state.deviceState = EC_DEVICE_STATE_OP);
    bExecute := FALSE;
END_IF
END_METHOD

PROPERTY PUBLIC EcatOk : BOOL
GET
EcatOk := _ecatOk;
END_GET
END_PROPERTY

PROPERTY PUBLIC ErrorTime : TIME
GET
ErrorTime := _errorTime;
END_GET
SET
_errorTime := ErrorTime;
END_SET
END_PROPERTY

METHOD PUBLIC ChangeState : BOOL
VAR_INPUT
    RequestedDeviceState : BYTE;
END_VAR
ChangeState := FALSE;

_setSlaveState(sNetId := _netId,
    nSlaveAddr := _etherCAT_Addr,
    bExecute :=,
    tTimeout :=,
    reqState :=,
    bBusy =>,
    bError =>,
    nErrId =>,
    currState => state);

CASE _progress OF
    0:
        _ecatOk := FALSE;
        _setSlaveState(bExecute := FALSE);
        _progress := 10;
    10:
        _setSlaveState(reqState := EC_DEVICE_STATE_INIT);
        _setSlaveState(bExecute := TRUE);

        IF _setSlaveState.bBusy THEN
            _progress := 15;
        END_IF
    15: //INIT
        IF (state.deviceState) = EC_DEVICE_STATE_INIT AND
            RequestedDeviceState > state.deviceState AND
            RequestedDeviceState <> EC_DEVICE_STATE_BOOTSTRAP THEN
            _setSlaveState(bExecute := FALSE);
            _progress := 30;
        ELSIF (state.deviceState) = EC_DEVICE_STATE_INIT AND
            RequestedDeviceState > state.deviceState AND
            RequestedDeviceState = EC_DEVICE_STATE_BOOTSTRAP THEN
            _setSlaveState(bExecute := FALSE);
            _progress := 20;
        ELSIF NOT _setSlaveState.bBusy AND (state.deviceState) = RequestedDeviceState THEN
            _progress := 100;
        END_IF
    20:
        _setSlaveState(reqState := EC_DEVICE_STATE_BOOTSTRAP);
        _setSlaveState(bExecute := TRUE);

        IF _setSlaveState.bBusy THEN
            _progress := 25;
        END_IF
    25: ///BOOTSTRAP
        IF (state.deviceState) = EC_DEVICE_STATE_BOOTSTRAP THEN
            _setSlaveState(bExecute := FALSE);
            _progress := 100;
        END_IF
    30:
        _setSlaveState(reqState := EC_DEVICE_STATE_PREOP);
        _setSlaveState(bExecute := TRUE);

        IF _setSlaveState.bBusy THEN
            _progress := 35;
        END_IF
    35: //PREOP
        IF (state.deviceState) = EC_DEVICE_STATE_PREOP AND RequestedDeviceState > state.deviceState THEN
            _setSlaveState(bExecute := FALSE);
            _progress := 40;
        ELSIF NOT _setSlaveState.bBusy AND (state.deviceState) = RequestedDeviceState THEN
            _progress := 100;
        END_IF
    40:
        _setSlaveState(reqState := EC_DEVICE_STATE_SAFEOP);
        _setSlaveState(bExecute := TRUE);

        IF _setSlaveState.bBusy THEN
            _progress := 45;
        END_IF
    45: //SAFEOP
        IF (state.deviceState) = EC_DEVICE_STATE_SAFEOP AND RequestedDeviceState > state.deviceState THEN
            _setSlaveState(bExecute := FALSE);
            _progress := 50;
        ELSIF NOT _setSlaveState.bBusy AND (state.deviceState) = RequestedDeviceState THEN
            _progress := 100;
        END_IF
    50: //OP
        _setSlaveState(reqState := EC_DEVICE_STATE_OP);
        _setSlaveState(bExecute := TRUE);

        IF (state.deviceState) = EC_DEVICE_STATE_OP THEN
            _setSlaveState(bExecute := FALSE);
            _ecatOk := TRUE;
            _progress := 100;
        END_IF
    100:
        ChangeState := TRUE;
        _progress := 0;
END_CASE

Messenger.OnCondition(NOT _setSlaveState.bBusy AND RequestedDeviceState > EC_DEVICE_STATE_OP)
    .Post(_sb.Clear().Append('<#Unexpected state: #>').Append(TO_STRING(state.deviceState)).ToString(), eMessageCategory.Error);
END_METHOD

PROPERTY PUBLIC ChangeStateTask : TcoCore.ITcoTaskStatus
GET
ChangeStateTask := _changeStateTask;
END_GET
END_PROPERTY

PROPERTY PUBLIC PeriodCheckState : TIME
GET
PeriodCheckState := _periodStateCheckTime;
END_GET
SET
_periodStateCheckTime := PeriodCheckState;
END_SET
END_PROPERTY

METHOD Restore : ITcoRestorable
VAR_INPUT
END_VAR
_changeStateTask.Restore();
_ecatOk := false;
_progress := 0;
_restoreTask.Restore();
END_METHOD

END_FUNCTION_BLOCK

// ---- EtherCAT/TcoEcatComponent.TcPOU
FUNCTION_BLOCK ABSTRACT TcoEcatComponent EXTENDS TcoCore.TcoComponent IMPLEMENTS ITcoEcatComponent
VAR_INPUT
    AdsAddr : AMSADDR;
END_VAR
VAR_OUTPUT
END_VAR
VAR
    //*	{attribute addProperty Name "<#Ecat slave state#>"}
    _ecatState : TcoEcatSlaveState(THIS^);
    {attribute 'hide'}
    _sb : TcoCore.StringBuilder;
END_VAR

_ecatState(AdsAddr := AdsAddr);

PROPERTY PUBLIC EcatState : REFERENCE TO TcoEcatSlaveState
GET
EcatState REF= _ecatState;
END_GET
END_PROPERTY

METHOD Restore : ITcoRestorable
VAR_INPUT
END_VAR
_ecatState.Restore();
END_METHOD

METHOD PROTECTED ServiceMode
VAR_INPUT
END_VAR
END_METHOD

END_FUNCTION_BLOCK
